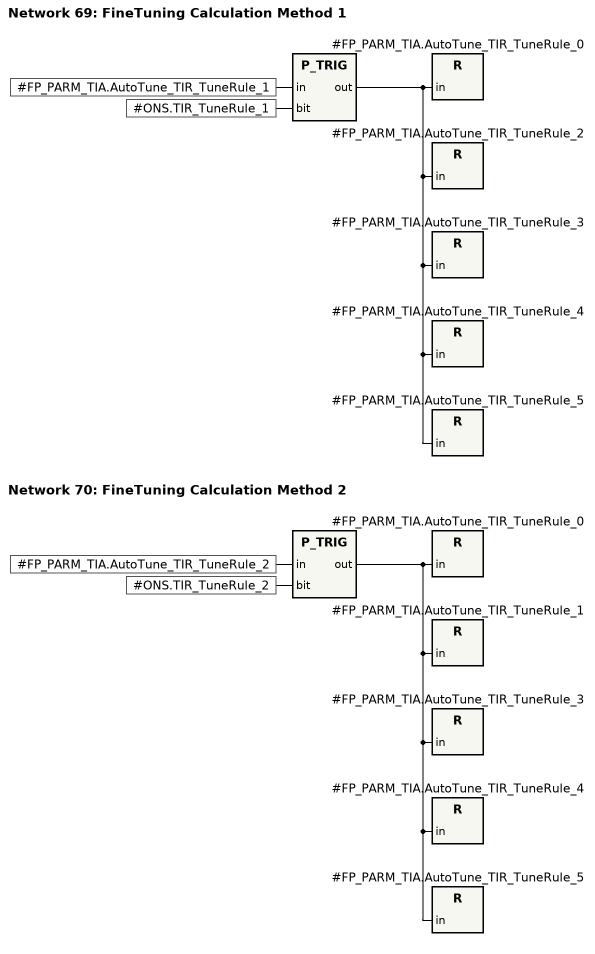
   #_w1 := #FP_PARM_TIA.AutoTune_TIR_TuneRule_1 AND NOT #ONS.TIR_TuneRule_1;   // rising edge
   #ONS.TIR_TuneRule_1 := #FP_PARM_TIA.AutoTune_TIR_TuneRule_1;
   IF #_w1 THEN
       #FP_PARM_TIA.AutoTune_TIR_TuneRule_0 := FALSE;
       #FP_PARM_TIA.AutoTune_TIR_TuneRule_2 := FALSE;
       #FP_PARM_TIA.AutoTune_TIR_TuneRule_3 := FALSE;
       #FP_PARM_TIA.AutoTune_TIR_TuneRule_4 := FALSE;
       #FP_PARM_TIA.AutoTune_TIR_TuneRule_5 := FALSE;
   END_IF;
END_REGION

REGION Network 70: FineTuning Calculation Method 2
   #_w1 := #FP_PARM_TIA.AutoTune_TIR_TuneRule_2 AND NOT #ONS.TIR_TuneRule_2;   // rising edge
   #ONS.TIR_TuneRule_2 := #FP_PARM_TIA.AutoTune_TIR_TuneRule_2;
   IF #_w1 THEN
       #FP_PARM_TIA.AutoTune_TIR_TuneRule_0 := FALSE;
       #FP_PARM_TIA.AutoTune_TIR_TuneRule_1 := FALSE;
       #FP_PARM_TIA.AutoTune_TIR_TuneRule_3 := FALSE;
       #FP_PARM_TIA.AutoTune_TIR_TuneRule_4 := FALSE;
       #FP_PARM_TIA.AutoTune_TIR_TuneRule_5 := FALSE;
   END_IF;
END_REGION

REGION Network 71: FineTuning Calculation Method 3
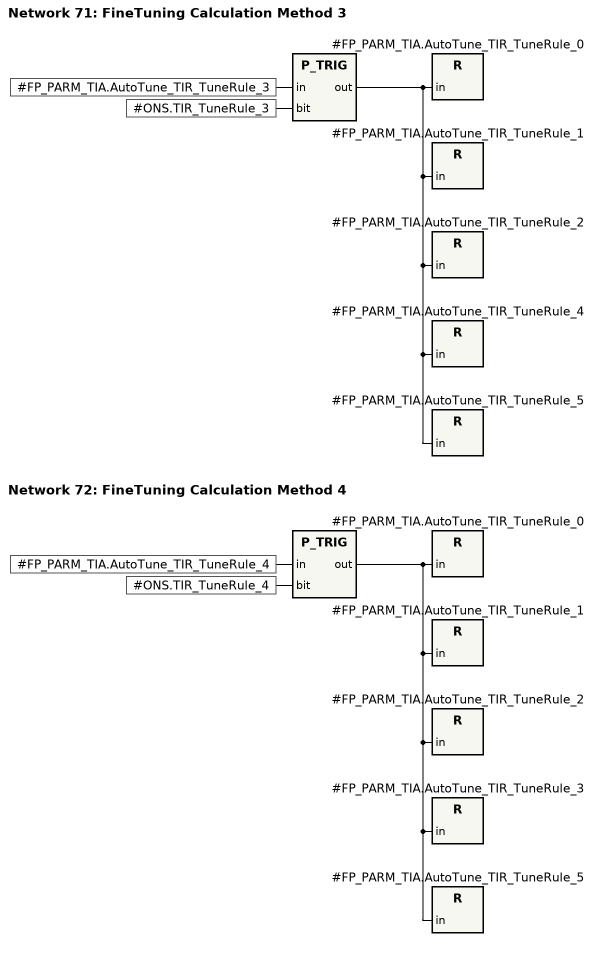
   #_w1 := #FP_PARM_TIA.AutoTune_TIR_TuneRule_3 AND NOT #ONS.TIR_TuneRule_3;   // rising edge
   #ONS.TIR_TuneRule_3 := #FP_PARM_TIA.AutoTune_TIR_TuneRule_3;
   IF #_w1 THEN
       #FP_PARM_TIA.AutoTune_TIR_TuneRule_0 := FALSE;
       #FP_PARM_TIA.AutoTune_TIR_TuneRule_1 := FALSE;
       #FP_PARM_TIA.AutoTune_TIR_TuneRule_2 := FALSE;
       #FP_PARM_TIA.AutoTune_TIR_TuneRule_4 := FALSE;
       #FP_PARM_TIA.AutoTune_TIR_TuneRule_5 := FALSE;
   END_IF;
END_REGION

REGION Network 72: FineTuning Calculation Method 4
   #_w1 := #FP_PARM_TIA.AutoTune_TIR_TuneRule_4 AND NOT #ONS.TIR_TuneRule_4;   // rising edge
   #ONS.TIR_TuneRule_4 := #FP_PARM_TIA.AutoTune_TIR_TuneRule_4;
   IF #_w1 THEN
       #FP_PARM_TIA.AutoTune_TIR_TuneRule_0 := FALSE;
       #FP_PARM_TIA.AutoTune_TIR_TuneRule_1 := FALSE;
       #FP_PARM_TIA.AutoTune_TIR_TuneRule_2 := FALSE;
       #FP_PARM_TIA.AutoTune_TIR_TuneRule_3 := FALSE;
       #FP_PARM_TIA.AutoTune_TIR_TuneRule_5 := FALSE;
   END_IF;
END_REGION

REGION Network 73: FineTuning Calculation Method 5
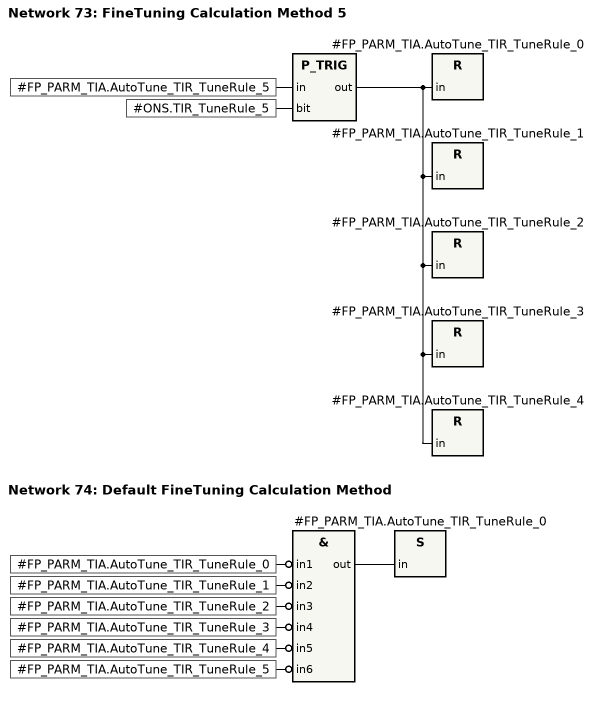
   #_w1 := #FP_PARM_TIA.AutoTune_TIR_TuneRule_5 AND NOT #ONS.TIR_TuneRule_5;   // rising edge
   #ONS.TIR_TuneRule_5 := #FP_PARM_TIA.AutoTune_TIR_TuneRule_5;
   IF #_w1 THEN
       #FP_PARM_TIA.AutoTune_TIR_TuneRule_0 := FALSE;
       #FP_PARM_TIA.AutoTune_TIR_TuneRule_1 := FALSE;
       #FP_PARM_TIA.AutoTune_TIR_TuneRule_2 := FALSE;
       #FP_PARM_TIA.AutoTune_TIR_TuneRule_3 := FALSE;
       #FP_PARM_TIA.AutoTune_TIR_TuneRule_4 := FALSE;
   END_IF;
END_REGION

REGION Network 74: Default FineTuning Calculation Method
   IF NOT #FP_PARM_TIA.AutoTune_TIR_TuneRule_0 AND NOT #FP_PARM_TIA.AutoTune_TIR_TuneRule_1 AND NOT #FP_PARM_TIA.AutoTune_TIR_TuneRule_2 AND NOT #FP_PARM_TIA.AutoTune_TIR_TuneRule_3 AND NOT #FP_PARM_TIA.AutoTune_TIR_TuneRule_4 AND NOT #FP_PARM_TIA.AutoTune_TIR_TuneRule_5 THEN
       #FP_PARM_TIA.AutoTune_TIR_TuneRule_0 := TRUE;
   END_IF;
END_REGION

REGION Network 75: AutoTune Parameterization
   // Build 002 - 04. Mar 2019 (RULA) : Typo in Auto tuning methods definition is corrected
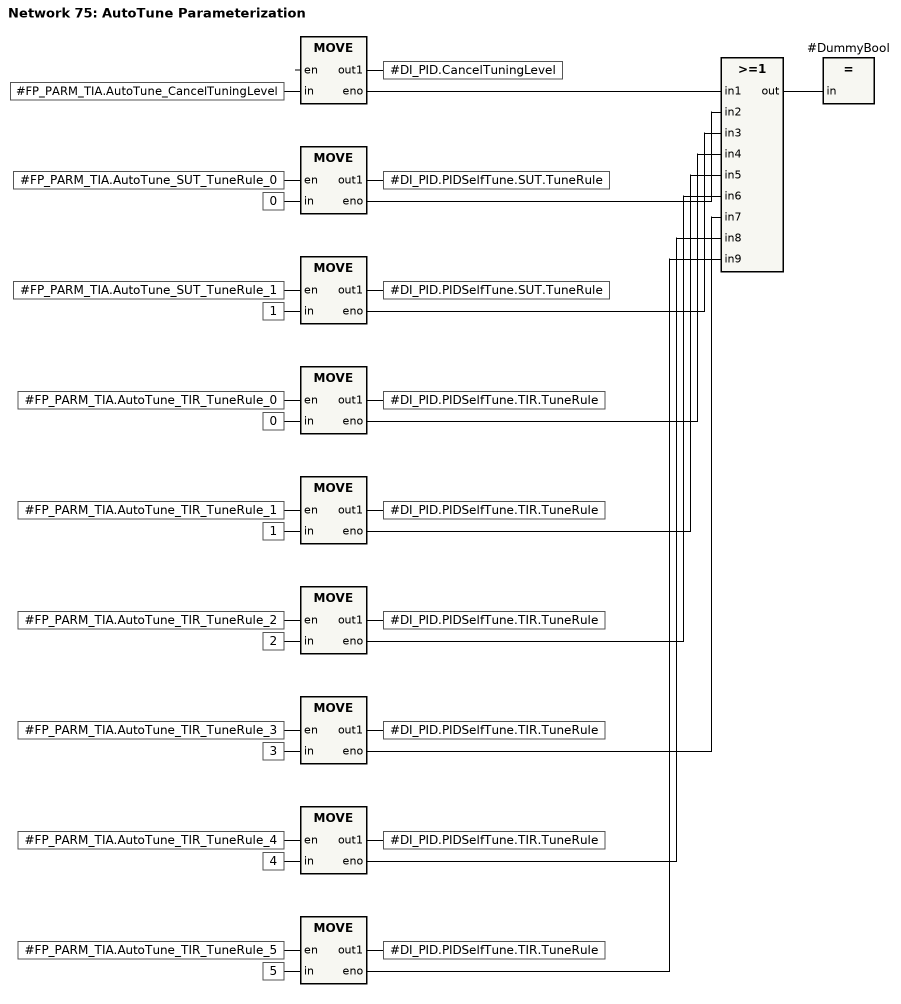
   #DI_PID.CancelTuningLevel := #FP_PARM_TIA.AutoTune_CancelTuningLevel;
   IF #FP_PARM_TIA.AutoTune_SUT_TuneRule_0 THEN #DI_PID.PIDSelfTune.SUT.TuneRule := 0; END_IF;
   IF #FP_PARM_TIA.AutoTune_SUT_TuneRule_1 THEN #DI_PID.PIDSelfTune.SUT.TuneRule := 1; END_IF;
   IF #FP_PARM_TIA.AutoTune_TIR_TuneRule_0 THEN #DI_PID.PIDSelfTune.TIR.TuneRule := 0; END_IF;
   IF #FP_PARM_TIA.AutoTune_TIR_TuneRule_1 THEN #DI_PID.PIDSelfTune.TIR.TuneRule := 1; END_IF;
   IF #FP_PARM_TIA.AutoTune_TIR_TuneRule_2 THEN #DI_PID.PIDSelfTune.TIR.TuneRule := 2; END_IF;
   IF #FP_PARM_TIA.AutoTune_TIR_TuneRule_3 THEN #DI_PID.PIDSelfTune.TIR.TuneRule := 3; END_IF;
   IF #FP_PARM_TIA.AutoTune_TIR_TuneRule_4 THEN #DI_PID.PIDSelfTune.TIR.TuneRule := 4; END_IF;
   IF #FP_PARM_TIA.AutoTune_TIR_TuneRule_5 THEN #DI_PID.PIDSelfTune.TIR.TuneRule := 5; END_IF;
   #DummyBool := TRUE OR #FP_PARM_TIA.AutoTune_SUT_TuneRule_0 OR #FP_PARM_TIA.AutoTune_SUT_TuneRule_1 OR #FP_PARM_TIA.AutoTune_TIR_TuneRule_0 OR #FP_PARM_TIA.AutoTune_TIR_TuneRule_1 OR #FP_PARM_TIA.AutoTune_TIR_TuneRule_2 OR #FP_PARM_TIA.AutoTune_TIR_TuneRule_3 OR #FP_PARM_TIA.AutoTune_TIR_TuneRule_4 OR #FP_PARM_TIA.AutoTune_TIR_TuneRule_5;
END_REGION

REGION Network 76: PreTuning Phase
   // 0: Initialize PreTuning
   // 100: Calculate Standard Deviation
   // 200: Find Point of Inflection
   // 9900: PreTuning Succesful
   // 1: PreTuning not Succesful
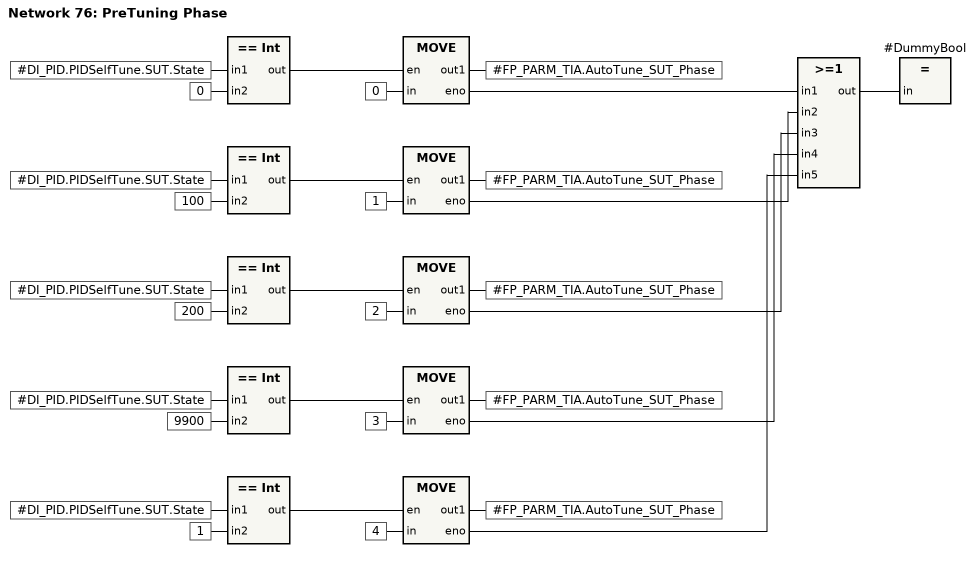
   #_w1 := #DI_PID.PIDSelfTune.SUT.State = 0;
   IF #_w1 THEN #FP_PARM_TIA.AutoTune_SUT_Phase := 0; END_IF;
   #_w2 := #DI_PID.PIDSelfTune.SUT.State = 100;
   IF #_w2 THEN #FP_PARM_TIA.AutoTune_SUT_Phase := 1; END_IF;
   #_w3 := #DI_PID.PIDSelfTune.SUT.State = 200;
   IF #_w3 THEN #FP_PARM_TIA.AutoTune_SUT_Phase := 2; END_IF;
   #_w4 := #DI_PID.PIDSelfTune.SUT.State = 9900;
   IF #_w4 THEN #FP_PARM_TIA.AutoTune_SUT_Phase := 3; END_IF;
   #_w5 := #DI_PID.PIDSelfTune.SUT.State = 1;
   IF #_w5 THEN #FP_PARM_TIA.AutoTune_SUT_Phase := 4; END_IF;
   #DummyBool := #_w1 OR #_w2 OR #_w3 OR #_w4 OR #_w5;
END_REGION

REGION Network 77: FineTuning Phase
   // -100: FineTuning not Possible.  PreTuning first
   // 0: Initialize FineTuning
   // 200:Calculate Standard Deviation
   // 300: Attempt to Reach Setpoint
   // 400: Attempt to Reach Sepoint with existing PID parameters
   // 500: Determine Oscillation and Calculate Parameters
   // 9900: FineTuning Success
   // 1: FineTuning not Succesful
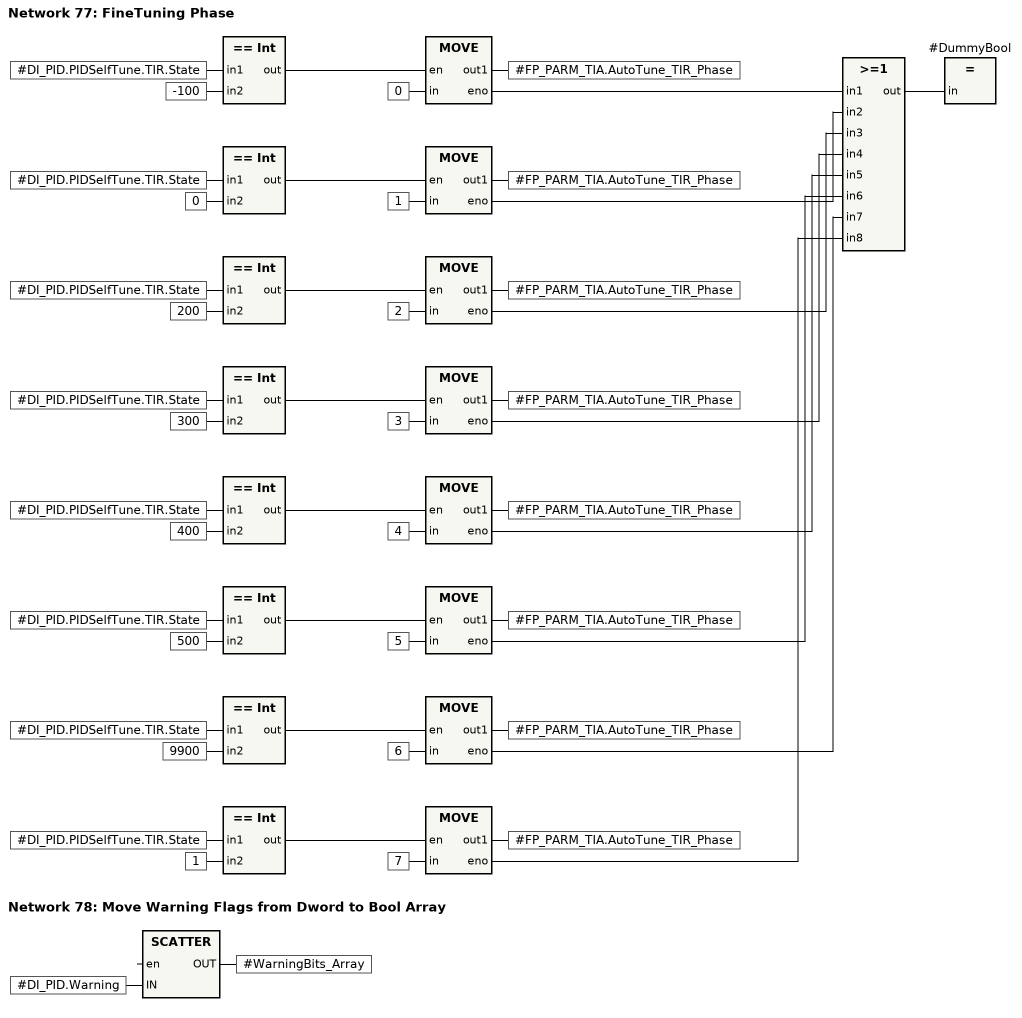
   #_w1 := #DI_PID.PIDSelfTune.TIR.State = (-100);
   IF #_w1 THEN #FP_PARM_TIA.AutoTune_TIR_Phase := 0; END_IF;
   #_w2 := #DI_PID.PIDSelfTune.TIR.State = 0;
   IF #_w2 THEN #FP_PARM_TIA.AutoTune_TIR_Phase := 1; END_IF;
   #_w3 := #DI_PID.PIDSelfTune.TIR.State = 200;
   IF #_w3 THEN #FP_PARM_TIA.AutoTune_TIR_Phase := 2; END_IF;
   #_w4 := #DI_PID.PIDSelfTune.TIR.State = 300;
   IF #_w4 THEN #FP_PARM_TIA.AutoTune_TIR_Phase := 3; END_IF;
   #_w5 := #DI_PID.PIDSelfTune.TIR.State = 400;
   IF #_w5 THEN #FP_PARM_TIA.AutoTune_TIR_Phase := 4; END_IF;
   #_w6 := #DI_PID.PIDSelfTune.TIR.State = 500;
   IF #_w6 THEN #FP_PARM_TIA.AutoTune_TIR_Phase := 5; END_IF;
   #_w7 := #DI_PID.PIDSelfTune.TIR.State = 9900;
   IF #_w7 THEN #FP_PARM_TIA.AutoTune_TIR_Phase := 6; END_IF;
   #_w8 := #DI_PID.PIDSelfTune.TIR.State = 1;
   IF #_w8 THEN #FP_PARM_TIA.AutoTune_TIR_Phase := 7; END_IF;
   #DummyBool := #_w1 OR #_w2 OR #_w3 OR #_w4 OR #_w5 OR #_w6 OR #_w7 OR #_w8;
END_REGION

REGION Network 78: Move Warning Flags from Dword to Bool Array
   SCATTER(IN := #DI_PID.Warning, OUT => #WarningBits_Array);
END_REGION

REGION Network 79: Warning Flags
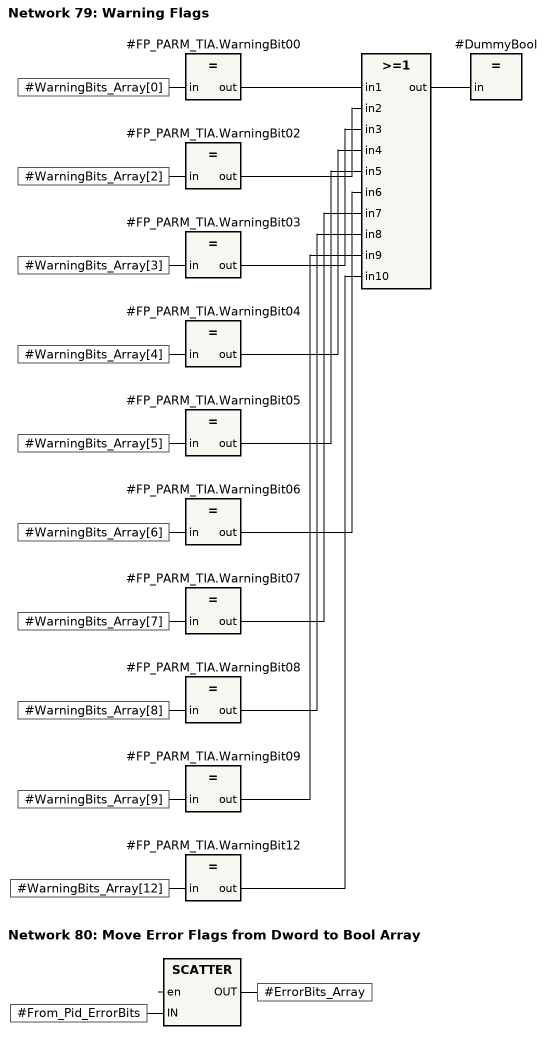
   #FP_PARM_TIA.WarningBit00 := #WarningBits_Array[0];
   #FP_PARM_TIA.WarningBit02 := #WarningBits_Array[2];
   #FP_PARM_TIA.WarningBit03 := #WarningBits_Array[3];
   #FP_PARM_TIA.WarningBit04 := #WarningBits_Array[4];
   #FP_PARM_TIA.WarningBit05 := #WarningBits_Array[5];
   #FP_PARM_TIA.WarningBit06 := #WarningBits_Array[6];
   #FP_PARM_TIA.WarningBit07 := #WarningBits_Array[7];
   #FP_PARM_TIA.WarningBit08 := #WarningBits_Array[8];
   #FP_PARM_TIA.WarningBit09 := #WarningBits_Array[9];
   #FP_PARM_TIA.WarningBit12 := #WarningBits_Array[12];
   #DummyBool := #WarningBits_Array[0] OR #WarningBits_Array[2] OR #WarningBits_Array[3] OR #WarningBits_Array[4] OR #WarningBits_Array[5] OR #WarningBits_Array[6] OR #WarningBits_Array[7] OR #WarningBits_Array[8] OR #WarningBits_Array[9] OR #WarningBits_Array[12];
END_REGION

REGION Network 80: Move Error Flags from Dword to Bool Array
   SCATTER(IN := #From_Pid_ErrorBits, OUT => #ErrorBits_Array);
END_REGION

REGION Network 81: Error Flags
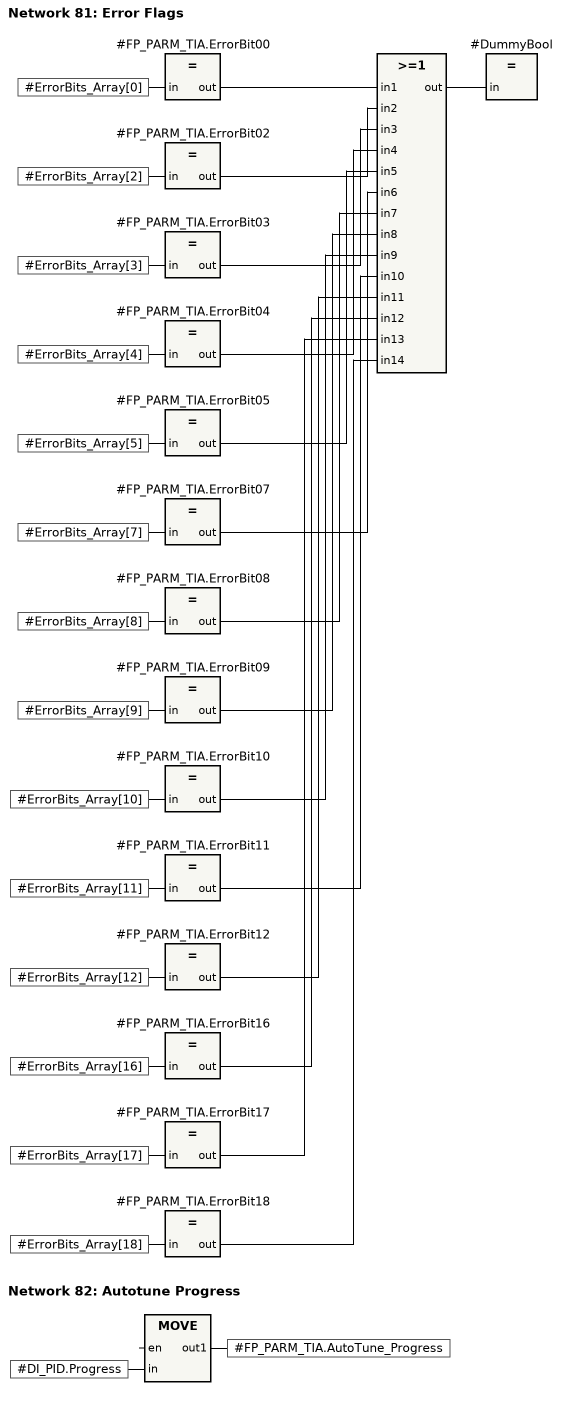
   #FP_PARM_TIA.ErrorBit00 := #ErrorBits_Array[0];
   #FP_PARM_TIA.ErrorBit02 := #ErrorBits_Array[2];
   #FP_PARM_TIA.ErrorBit03 := #ErrorBits_Array[3];
   #FP_PARM_TIA.ErrorBit04 := #ErrorBits_Array[4];
   #FP_PARM_TIA.ErrorBit05 := #ErrorBits_Array[5];
   #FP_PARM_TIA.ErrorBit07 := #ErrorBits_Array[7];
   #FP_PARM_TIA.ErrorBit08 := #ErrorBits_Array[8];
   #FP_PARM_TIA.ErrorBit09 := #ErrorBits_Array[9];
   #FP_PARM_TIA.ErrorBit10 := #ErrorBits_Array[10];
   #FP_PARM_TIA.ErrorBit11 := #ErrorBits_Array[11];
   #FP_PARM_TIA.ErrorBit12 := #ErrorBits_Array[12];
   #FP_PARM_TIA.ErrorBit16 := #ErrorBits_Array[16];
   #FP_PARM_TIA.ErrorBit17 := #ErrorBits_Array[17];
   #FP_PARM_TIA.ErrorBit18 := #ErrorBits_Array[18];
   #DummyBool := #ErrorBits_Array[0] OR #ErrorBits_Array[2] OR #ErrorBits_Array[3] OR #ErrorBits_Array[4] OR #ErrorBits_Array[5] OR #ErrorBits_Array[7] OR #ErrorBits_Array[8] OR #ErrorBits_Array[9] OR #ErrorBits_Array[10] OR #ErrorBits_Array[11] OR #ErrorBits_Array[12] OR #ErrorBits_Array[16] OR #ErrorBits_Array[17] OR #ErrorBits_Array[18];
END_REGION

REGION Network 82: Autotune Progress
   #FP_PARM_TIA.AutoTune_Progress := #DI_PID.Progress;
END_REGION

REGION Network 83: Update SPM Normalized
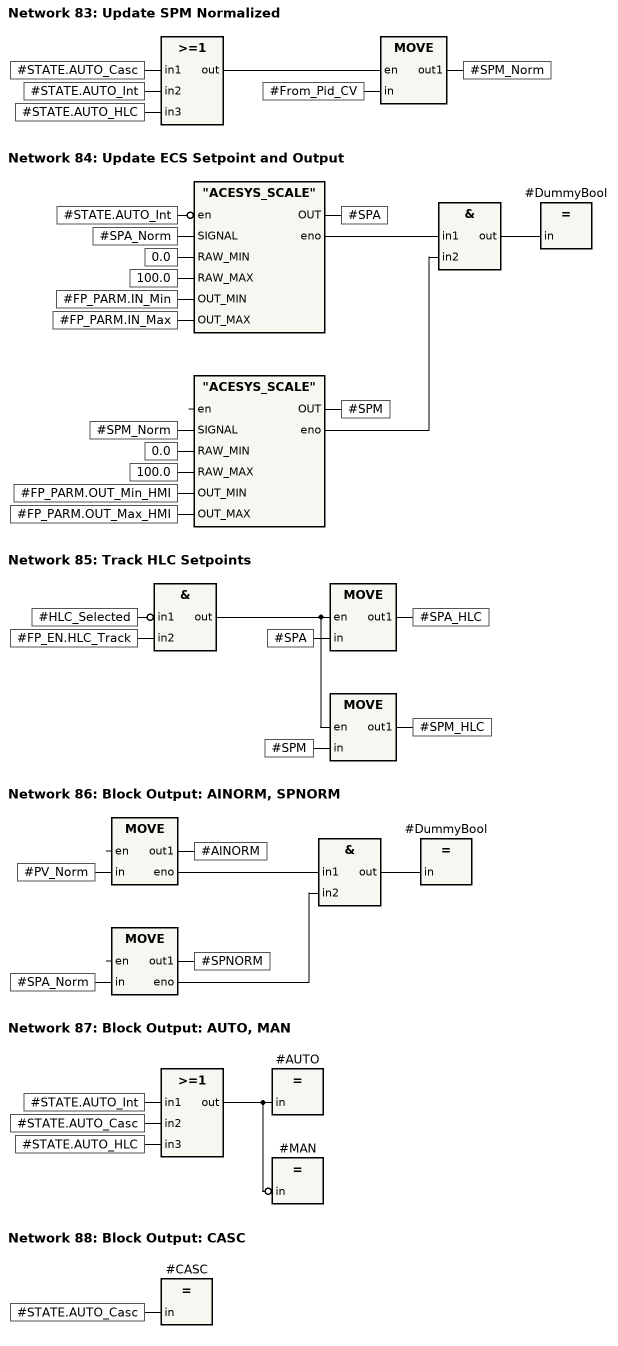
   IF #STATE.AUTO_Casc OR #STATE.AUTO_Int OR #STATE.AUTO_HLC THEN #SPM_Norm := #From_Pid_CV; END_IF;
END_REGION

REGION Network 84: Update ECS Setpoint and Output
   "ACESYS_SCALE"(EN := NOT #STATE.AUTO_Int,
                  SIGNAL := #SPA_Norm,
                  RAW_MIN := 0.0,
                  RAW_MAX := 100.0,
                  OUT_MIN := #FP_PARM.IN_Min,
                  OUT_MAX := #FP_PARM.IN_Max,
                  OUT => #SPA,
                  ENO => #_w1);
   "ACESYS_SCALE"(SIGNAL := #SPM_Norm,
                  RAW_MIN := 0.0,
                  RAW_MAX := 100.0,
                  OUT_MIN := #FP_PARM.OUT_Min_HMI,
                  OUT_MAX := #FP_PARM.OUT_Max_HMI,
                  OUT => #SPM,
                  ENO => #_w2);
   #DummyBool := #_w1 AND #_w2;
END_REGION

REGION Network 85: Track HLC Setpoints
   IF NOT #HLC_Selected AND #FP_EN.HLC_Track THEN
       #SPA_HLC := #SPA;
       #SPM_HLC := #SPM;
   END_IF;
END_REGION

REGION Network 86: Block Output: AINORM, SPNORM
   // >>>>> BLOCK OUTPUT <<<<<
   // ENO of a box is taken as its EN; it also drops when the box reports an error
   #AINORM := #PV_Norm;
   #SPNORM := #SPA_Norm;
   #DummyBool := TRUE;
END_REGION

REGION Network 87: Block Output: AUTO, MAN
   #AUTO := #STATE.AUTO_Int OR #STATE.AUTO_Casc OR #STATE.AUTO_HLC;
   #MAN := NOT #AUTO;
END_REGION

REGION Network 88: Block Output: CASC
   #CASC := #STATE.AUTO_Casc;
END_REGION

REGION Network 89: Normalized Error
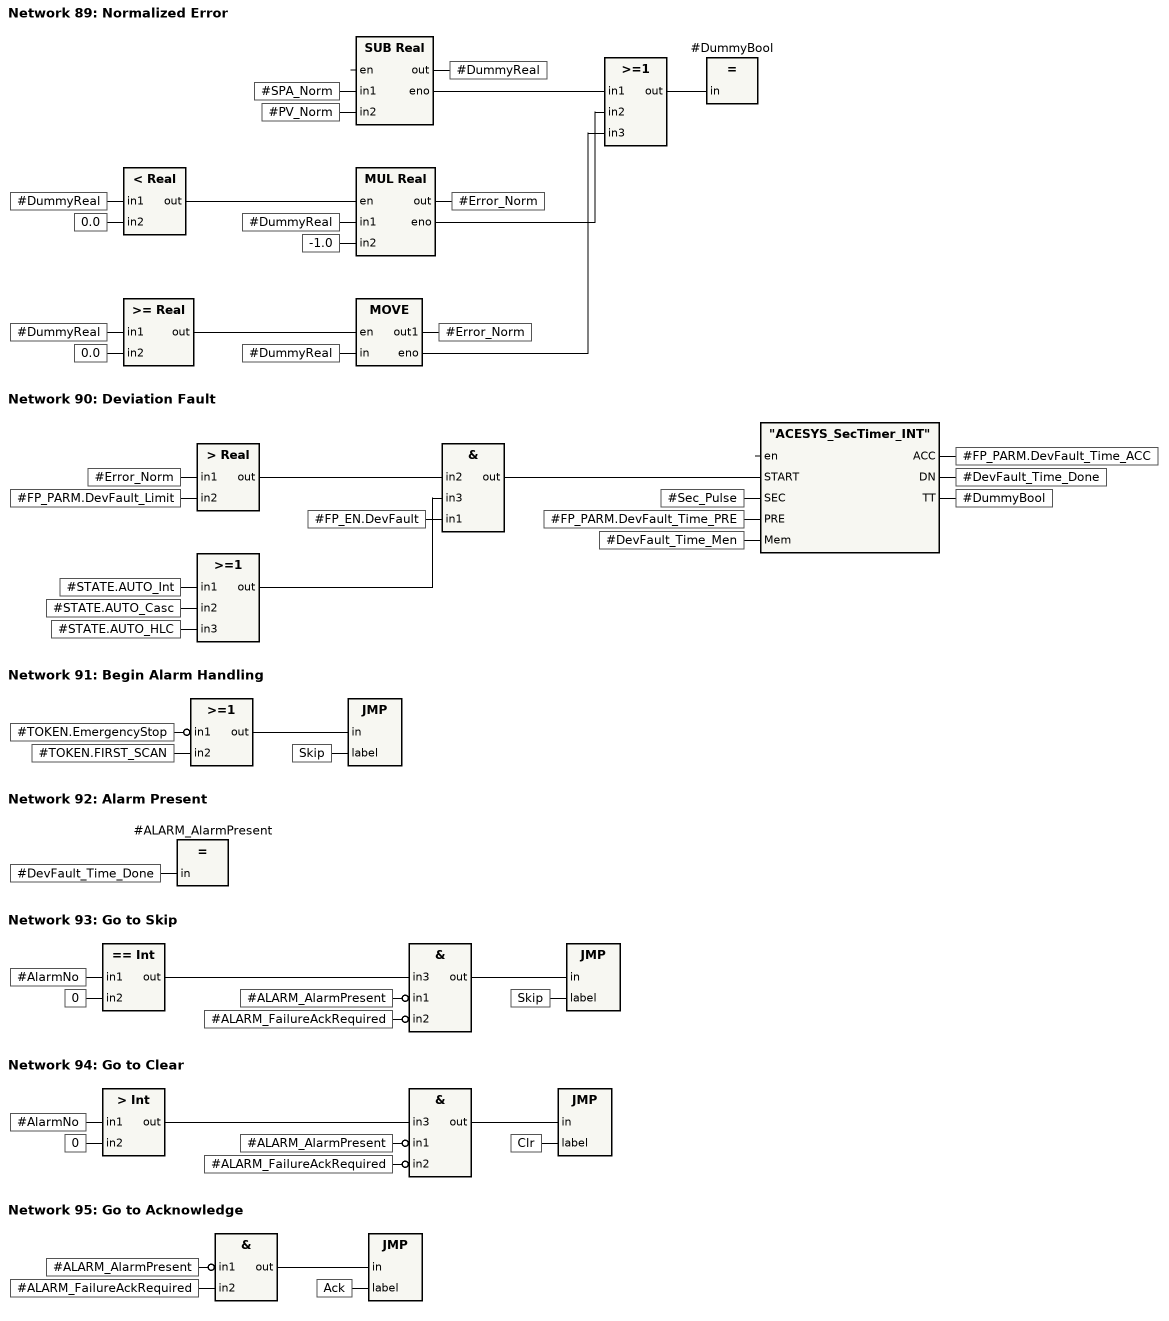
   #DummyReal := #SPA_Norm - #PV_Norm;
   #_w1 := #DummyReal < 0.0;
   IF #_w1 THEN #Error_Norm := #DummyReal * (-1.0); END_IF;
   #_w2 := #DummyReal >= 0.0;
   IF #_w2 THEN #Error_Norm := #DummyReal; END_IF;
   #DummyBool := TRUE OR #_w1 OR #_w2;
END_REGION

REGION Network 90: Deviation Fault
   // >>>>> DEVIATION FAULT <<<<<
   "ACESYS_SecTimer_INT"(START := (#Error_Norm > #FP_PARM.DevFault_Limit) AND (#STATE.AUTO_Int OR #STATE.AUTO_Casc OR #STATE.AUTO_HLC) AND #FP_EN.DevFault,
                         SEC := #Sec_Pulse,
                         PRE := #FP_PARM.DevFault_Time_PRE,
                         Mem := #DevFault_Time_Men,
                         ACC => #FP_PARM.DevFault_Time_ACC,
                         DN => #DevFault_Time_Done,
                         TT => #DummyBool);
END_REGION

REGION Network 91: Begin Alarm Handling
   // >>>>> ALARM HANDLING <<<<<
   IF NOT #TOKEN.EmergencyStop OR #TOKEN.FIRST_SCAN THEN GOTO Skip; END_IF;
END_REGION

REGION Network 92: Alarm Present
   #ALARM_AlarmPresent := #DevFault_Time_Done;
END_REGION

REGION Network 93: Go to Skip
   IF (#AlarmNo = 0) AND NOT #ALARM_AlarmPresent AND NOT #ALARM_FailureAckRequired THEN GOTO Skip; END_IF;
END_REGION

REGION Network 94: Go to Clear
   IF (#AlarmNo > 0) AND NOT #ALARM_AlarmPresent AND NOT #ALARM_FailureAckRequired THEN GOTO Clr; END_IF;
END_REGION

REGION Network 95: Go to Acknowledge
   IF NOT #ALARM_AlarmPresent AND #ALARM_FailureAckRequired THEN GOTO Ack; END_IF;
END_REGION

REGION Network 96: Alarm: Deviation Failure
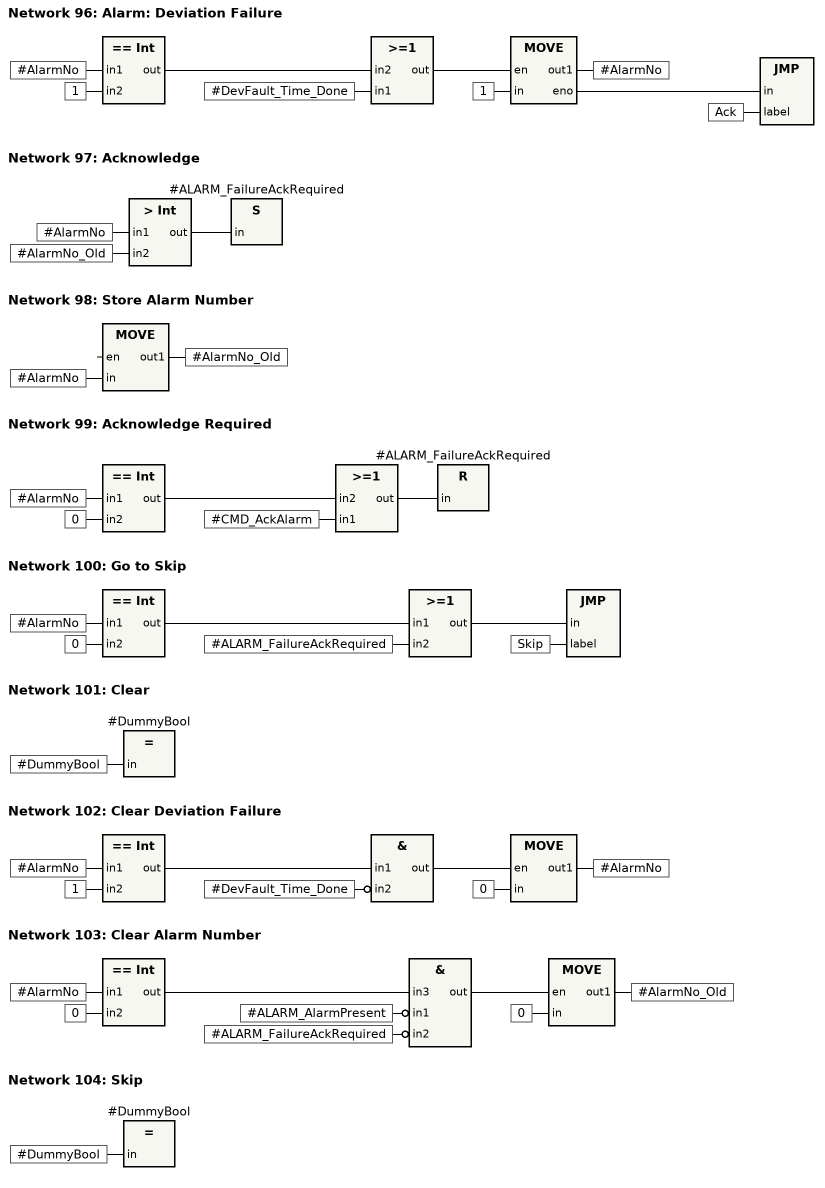
   // ENO of a box is taken as its EN; it also drops when the box reports an error
   #_w1 := (#AlarmNo = 1) OR #DevFault_Time_Done;
   IF #_w1 THEN
       #AlarmNo := 1;
       GOTO Ack;
   END_IF;
END_REGION

REGION Network 97: Acknowledge
   // ***Alarm Acknowledge***
   Ack:
   IF #AlarmNo > #AlarmNo_Old THEN #ALARM_FailureAckRequired := TRUE; END_IF;
END_REGION

REGION Network 98: Store Alarm Number
   #AlarmNo_Old := #AlarmNo;
END_REGION

REGION Network 99: Acknowledge Required
   IF (#AlarmNo = 0) OR #CMD_AckAlarm THEN #ALARM_FailureAckRequired := FALSE; END_IF;
END_REGION

REGION Network 100: Go to Skip
   IF (#AlarmNo = 0) OR #ALARM_FailureAckRequired THEN GOTO Skip; END_IF;
END_REGION

REGION Network 101: Clear
   Clr:
   #DummyBool := #DummyBool;
END_REGION

REGION Network 102: Clear Deviation Failure
   IF (#AlarmNo = 1) AND NOT #DevFault_Time_Done THEN #AlarmNo := 0; END_IF;
END_REGION

REGION Network 103: Clear Alarm Number
   IF (#AlarmNo = 0) AND NOT #ALARM_AlarmPresent AND NOT #ALARM_FailureAckRequired THEN
       #AlarmNo_Old := 0;
   END_IF;
END_REGION

REGION Network 104: Skip
   Skip:
   #DummyBool := #DummyBool;
END_REGION

REGION Network 105: Extended MSW
   // >>>> EXTENDED MSW to HMI <<<<<
   // 
   // Build 003 : 27. Jan. 2016 (FKP) : Network for #MSW.EXT.Operation changed from 
   //                                   AND- to OR-gate
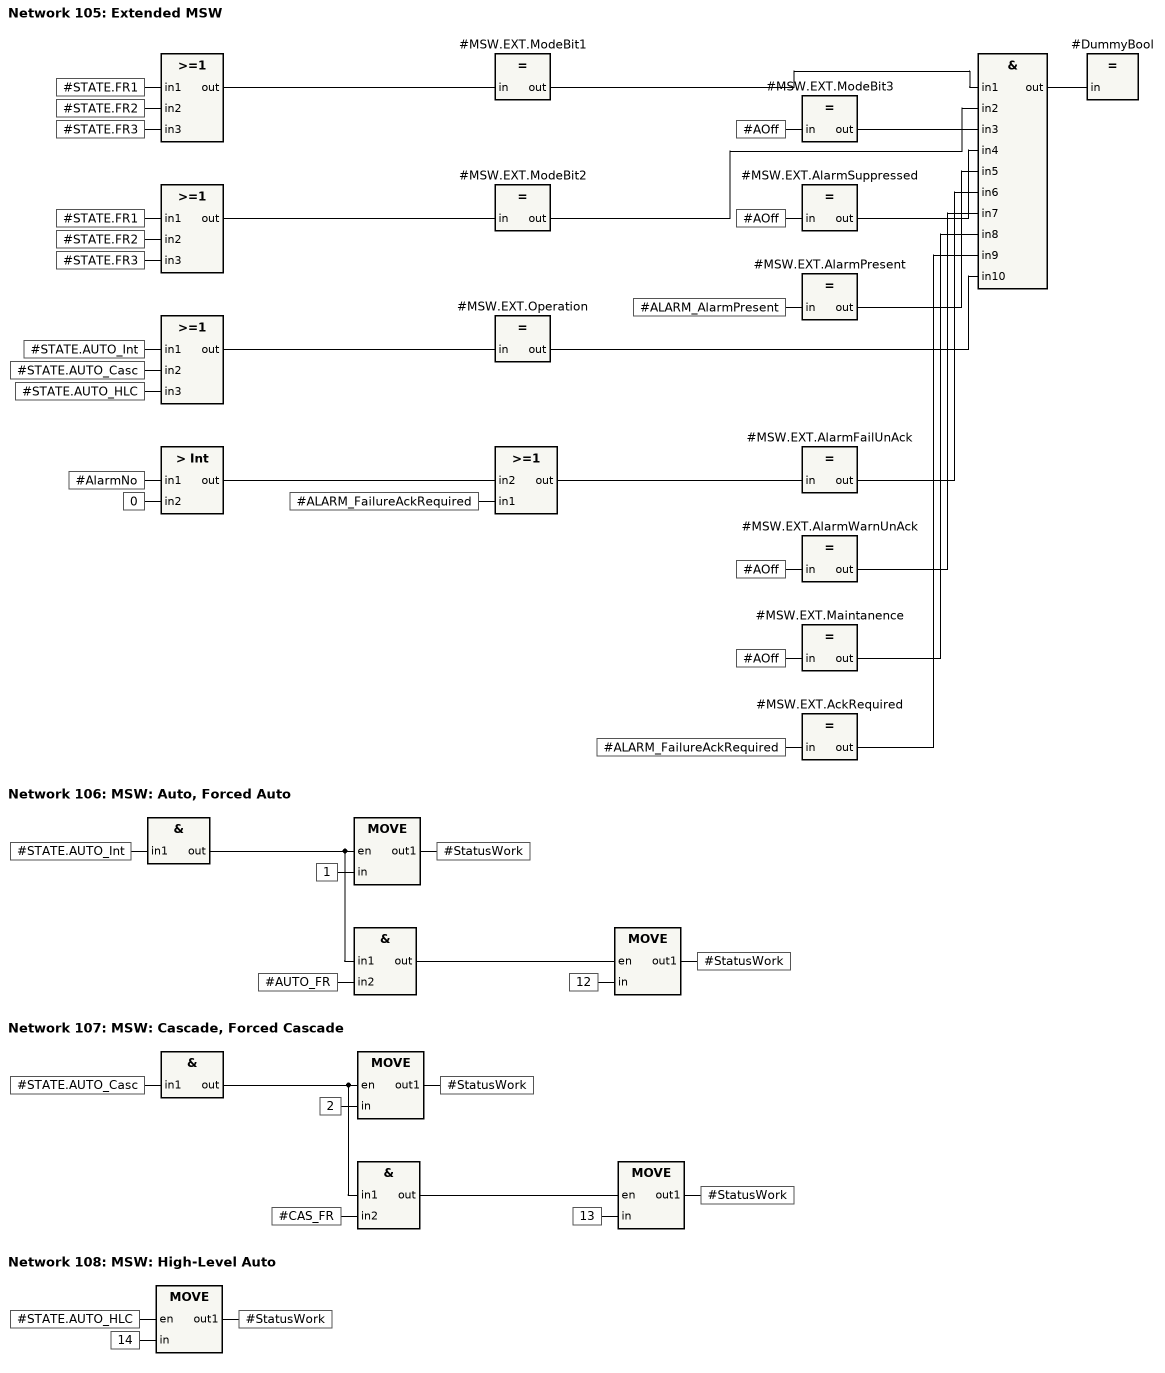
   #MSW.EXT.ModeBit1 := #STATE.FR1 OR #STATE.FR2 OR #STATE.FR3;
   #MSW.EXT.ModeBit2 := #STATE.FR1 OR #STATE.FR2 OR #STATE.FR3;
   #MSW.EXT.ModeBit3 := #AOff;
   #MSW.EXT.AlarmSuppressed := #AOff;
   #MSW.EXT.AlarmPresent := #ALARM_AlarmPresent;
   #MSW.EXT.AlarmFailUnAck := (#AlarmNo > 0) OR #ALARM_FailureAckRequired;
   #MSW.EXT.AlarmWarnUnAck := #AOff;
   #MSW.EXT.Maintanence := #AOff;
   #MSW.EXT.AckRequired := #ALARM_FailureAckRequired;
   #MSW.EXT.Operation := #STATE.AUTO_Int OR #STATE.AUTO_Casc OR #STATE.AUTO_HLC;
   #DummyBool := #MSW.EXT.ModeBit1 AND #MSW.EXT.ModeBit2 AND #AOff AND #AOff AND #ALARM_AlarmPresent AND #MSW.EXT.AlarmFailUnAck AND #AOff AND #AOff AND #ALARM_FailureAckRequired AND #MSW.EXT.Operation;
END_REGION

REGION Network 106: MSW: Auto, Forced Auto
   IF #STATE.AUTO_Int THEN #StatusWork := 1; END_IF;
   IF #STATE.AUTO_Int AND #AUTO_FR THEN #StatusWork := 12; END_IF;
END_REGION

REGION Network 107: MSW: Cascade, Forced Cascade
   IF #STATE.AUTO_Casc THEN #StatusWork := 2; END_IF;
   IF #STATE.AUTO_Casc AND #CAS_FR THEN #StatusWork := 13; END_IF;
END_REGION

REGION Network 108: MSW: High-Level Auto
   IF #STATE.AUTO_HLC THEN #StatusWork := 14; END_IF;
END_REGION

REGION Network 109: MSW: Manual, Forced Manual
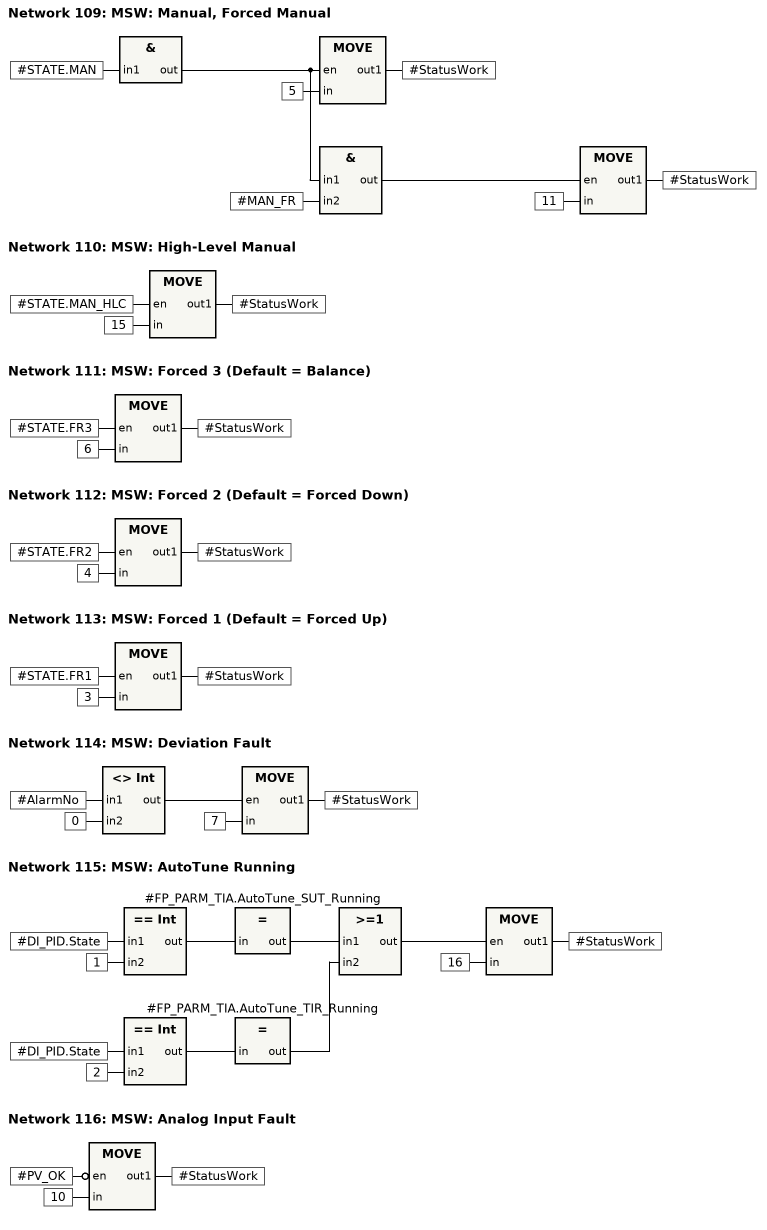
   IF #STATE.MAN THEN #StatusWork := 5; END_IF;
   IF #STATE.MAN AND #MAN_FR THEN #StatusWork := 11; END_IF;
END_REGION

REGION Network 110: MSW: High-Level Manual
   IF #STATE.MAN_HLC THEN #StatusWork := 15; END_IF;
END_REGION

REGION Network 111: MSW: Forced 3 (Default = Balance)
   IF #STATE.FR3 THEN #StatusWork := 6; END_IF;
END_REGION

REGION Network 112: MSW: Forced 2 (Default = Forced Down)
   IF #STATE.FR2 THEN #StatusWork := 4; END_IF;
END_REGION

REGION Network 113: MSW: Forced 1 (Default = Forced Up)
   IF #STATE.FR1 THEN #StatusWork := 3; END_IF;
END_REGION

REGION Network 114: MSW: Deviation Fault
   IF #AlarmNo <> 0 THEN #StatusWork := 7; END_IF;
END_REGION

REGION Network 115: MSW: AutoTune Running
   #FP_PARM_TIA.AutoTune_SUT_Running := #DI_PID.State = 1;
   #FP_PARM_TIA.AutoTune_TIR_Running := #DI_PID.State = 2;
   IF #FP_PARM_TIA.AutoTune_SUT_Running OR #FP_PARM_TIA.AutoTune_TIR_Running THEN #StatusWork := 16; END_IF;
END_REGION

REGION Network 116: MSW: Analog Input Fault
   IF NOT #PV_OK THEN #StatusWork := 10; END_IF;
END_REGION

REGION Network 117: Update Internal MSW and Timestamp
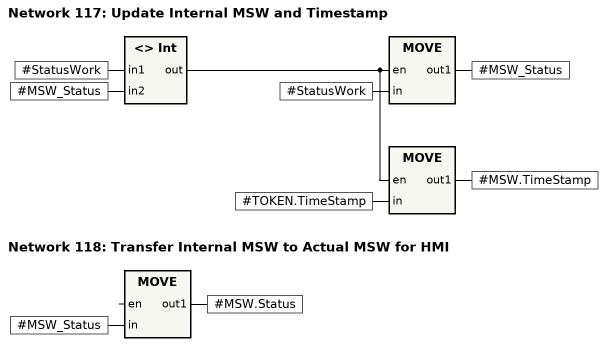
   #_w1 := #StatusWork <> #MSW_Status;
   IF #_w1 THEN
       #MSW_Status := #StatusWork;
       #MSW.TimeStamp := #TOKEN.TimeStamp;
   END_IF;
END_REGION

REGION Network 118: Transfer Internal MSW to Actual MSW for HMI
   #MSW.Status := #MSW_Status;
END_REGION
END_FUNCTION_BLOCK

FUNCTION_BLOCK "ACESYS_HLC"   // FB221, FBD
TITLE = ACESYS V8.0 - Build 001 - HIGH LEVEL CONTROL
{ S7_Optimized_Access := 'FALSE' }
AUTHOR : FLSmidth
FAMILY : ACESYS
NAME : HLC
VERSION : 8.0
   VAR_INPUT
      DEPT_LINK : "ACESYS_DEPT_LINK";   // Unit Number
      CCA1 : Bool := TRUE;   // Computer Control Accept Group 01-05
      CCA2 : Bool := TRUE;   // Computer Control Accept Group 06-10
      GRP_01_RDY : Bool := TRUE;   // Group 01 Ready
      GRP_02_RDY : Bool := TRUE;   // Group 02 Ready
      GRP_03_RDY : Bool := TRUE;   // Group 03 Ready
      GRP_04_RDY : Bool := TRUE;   // Group 04 Ready
      GRP_05_RDY : Bool := TRUE;   // Group 05 Ready
      GRP_06_RDY : Bool := TRUE;   // Group 06 Ready
      GRP_07_RDY : Bool := TRUE;   // Group 07 Ready
      GRP_08_RDY : Bool := TRUE;   // Group 08 Ready
      GRP_09_RDY : Bool := TRUE;   // Group 09 Ready
      GRP_10_RDY : Bool := TRUE;   // Group 10 Ready
   END_VAR
   VAR_OUTPUT
      HLC_LINK : "ACESYS_HLC_LINK";
      MSW : "ACESYS_HMI_STAT_32T";
   END_VAR
   VAR_IN_OUT
      KA : Bool;   // Keep Alive - Watchdog supervision
      GRP_01_EN : Bool;   // Enable Group 01
      GRP_02_EN : Bool;   // Enable Group 02
      GRP_03_EN : Bool;   // Enable Group 03
      GRP_04_EN : Bool;   // Enable Group 04
      GRP_05_EN : Bool;   // Enable Group 05
      GRP_06_EN : Bool;   // Enable Group 06
      GRP_07_EN : Bool;   // Enable Group 07
      GRP_08_EN : Bool;   // Enable Group 08
      GRP_09_EN : Bool;   // Enable Group 09
      GRP_10_EN : Bool;   // Enable Group 10
   END_VAR
   VAR
      BlockInfo : Struct
         Ace_Version : Int;   // Acesys Block Version Number
         Ace_BuildNo : Int;   // Acesys Block Build Number
         DB_Number : Int;   // Block Instance DB Number
      END_STRUCT;
      FP_CMD : Struct   // Faceplate Commands
         Spare_08 : Bool;
         Spare_09 : Bool;
         Spare_10 : Bool;
         Spare_11 : Bool;
         Spare_12 : Bool;
         Spare_13 : Bool;
         Spare_14 : Bool;
         AckAlarm : Bool;   // Alarm Acknowledge
         Spare_00 : Bool;
         Spare_01 : Bool;
         Spare_02 : Bool;
         Spare_03 : Bool;
         Spare_04 : Bool;
         Spare_05 : Bool;
         Spare_06 : Bool;
         Spare_07 : Bool;
      END_STRUCT;
      FP_SEL : Struct
         GRP_01 : Bool;
         GRP_02 : Bool;
         GRP_03 : Bool;
         GRP_04 : Bool;
         GRP_05 : Bool;
         GRP_06 : Bool;
         GRP_07 : Bool;
         GRP_08 : Bool;
         GRP_09 : Bool;
         GRP_10 : Bool;
         KA_Alarm : Bool;   // Select KA Supervision
         CCA1_Alarm : Bool;   // Select CCA Supervision HLC Group 01-05
         CCA2_Alarm : Bool;   // Select CCA Supervision HLC Group 06-10
         Spare3 : Bool;
         Spare2 : Bool;
         Spare1 : Bool;
      END_STRUCT;
      FP_EN : Struct
         Clear_Sel_CCA : Bool;   // Clear Selections when CCA Faults
         Clear_Sel_KA : Bool;   // Clear Selections when KA Fault
         Spare14 : Bool;
         Spare13 : Bool;
         Spare12 : Bool;
         Spare11 : Bool;
         Spare10 : Bool;
         Spare09 : Bool;
         Spare08 : Bool;
         Spare07 : Bool;
         Spare06 : Bool;
         Spare05 : Bool;
         Spare04 : Bool;
         Spare03 : Bool;
         Spare02 : Bool;
         Spare01 : Bool;
      END_STRUCT;
      FP_PARM : Struct
         KA_Time_Actual : Int;   // Keep Alive remaining time
         KA_Time_Setp : Int := 60;   // Keep Alive Setpoint
      END_STRUCT;
      ONS : Struct
         ONS_Off : Array[1..16] of Bool;
         ONS_On : Array[1..16] of Bool;
         OFF_01 : Bool;
         OFF_02 : Bool;
         OFF_03 : Bool;
         OFF_04 : Bool;
         OFF_05 : Bool;
         OFF_06 : Bool;
         OFF_07 : Bool;
         OFF_08 : Bool;
         OFF_09 : Bool;
         OFF_10 : Bool;
         ON_01 : Bool;
         ON_02 : Bool;
         ON_03 : Bool;
         ON_04 : Bool;
         ON_05 : Bool;
         ON_06 : Bool;
         ON_07 : Bool;
         ON_08 : Bool;
         ON_09 : Bool;
         ON_10 : Bool;
      END_STRUCT;
      KA_Time_Memory : Int;   // Keep Alive memory
      StatusToEcs : Int;
      ALARM_AlarmPresent : Bool;
      ALARM_FailureAckRequired : Bool;
      CMD_AckAlarm : Bool;
      StatusWork : Int;   // Internal Status Word
      AlarmNo : Int;
      AlarmNo_Old : Int;
      MSW_Status_Trans : Int;
   END_VAR
   VAR_TEMP
      Aon : Bool;
      Aoff : Bool;
      DummyBool : Bool;
      Acknowledge : Bool;   // Alarm Acknowledge
      KeepAliveTimeDone : Bool;
      TrigAlarm_KA : Bool;
      TrigAlarm_CCA1 : Bool;
      TrigAlarm_CCA2 : Bool;
   END_VAR
   VAR_TEMP   // added for the SCL form of the ladder/FBD networks
      _w1 : Bool;
   END_VAR
BEGIN

REGION Network 1: Always On
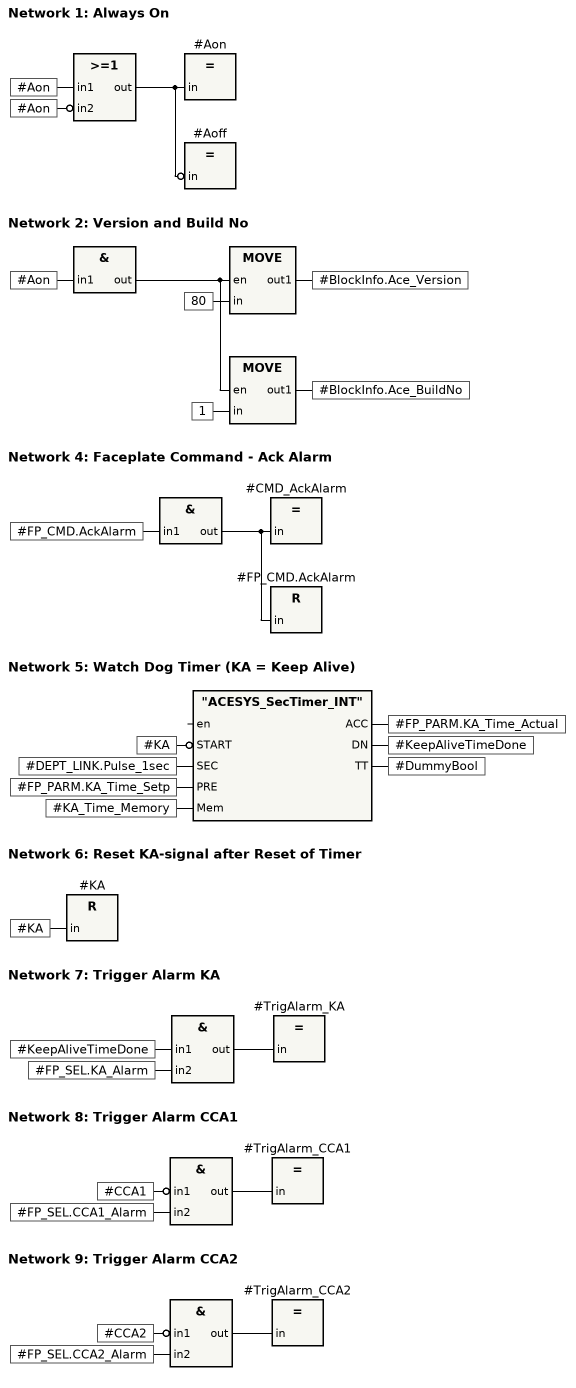
   #Aon := #Aon OR NOT #Aon;
   #Aoff := NOT #Aon;
END_REGION

REGION Network 2: Version and Build No
   IF #Aon THEN
       #BlockInfo.Ace_Version := 80;
       #BlockInfo.Ace_BuildNo := 1;
   END_IF;
END_REGION

REGION Network 3 (STL): Instance DB Number to Faceplate
         L     DINO;
         T     #BlockInfo.DB_Number;
END_REGION

REGION Network 4: Faceplate Command - Ack Alarm
   #CMD_AckAlarm := #FP_CMD.AckAlarm;
   IF #FP_CMD.AckAlarm THEN #FP_CMD.AckAlarm := FALSE; END_IF;
END_REGION

REGION Network 5: Watch Dog Timer (KA = Keep Alive)
   "ACESYS_SecTimer_INT"(START := NOT #KA,
                         SEC := #DEPT_LINK.Pulse_1sec,
                         PRE := #FP_PARM.KA_Time_Setp,
                         Mem := #KA_Time_Memory,
                         ACC => #FP_PARM.KA_Time_Actual,
                         DN => #KeepAliveTimeDone,
                         TT => #DummyBool);
END_REGION

REGION Network 6: Reset KA-signal after Reset of Timer
   IF #KA THEN #KA := FALSE; END_IF;
END_REGION

REGION Network 7: Trigger Alarm KA
   #TrigAlarm_KA := #KeepAliveTimeDone AND #FP_SEL.KA_Alarm;
END_REGION

REGION Network 8: Trigger Alarm CCA1
   #TrigAlarm_CCA1 := NOT #CCA1 AND #FP_SEL.CCA1_Alarm;
END_REGION

REGION Network 9: Trigger Alarm CCA2
   #TrigAlarm_CCA2 := NOT #CCA2 AND #FP_SEL.CCA2_Alarm;
END_REGION

REGION Network 10: If Intput is changed, Update Faceplate Parameters - Sel GRP01
   // >>>>> SELECT <<<<<
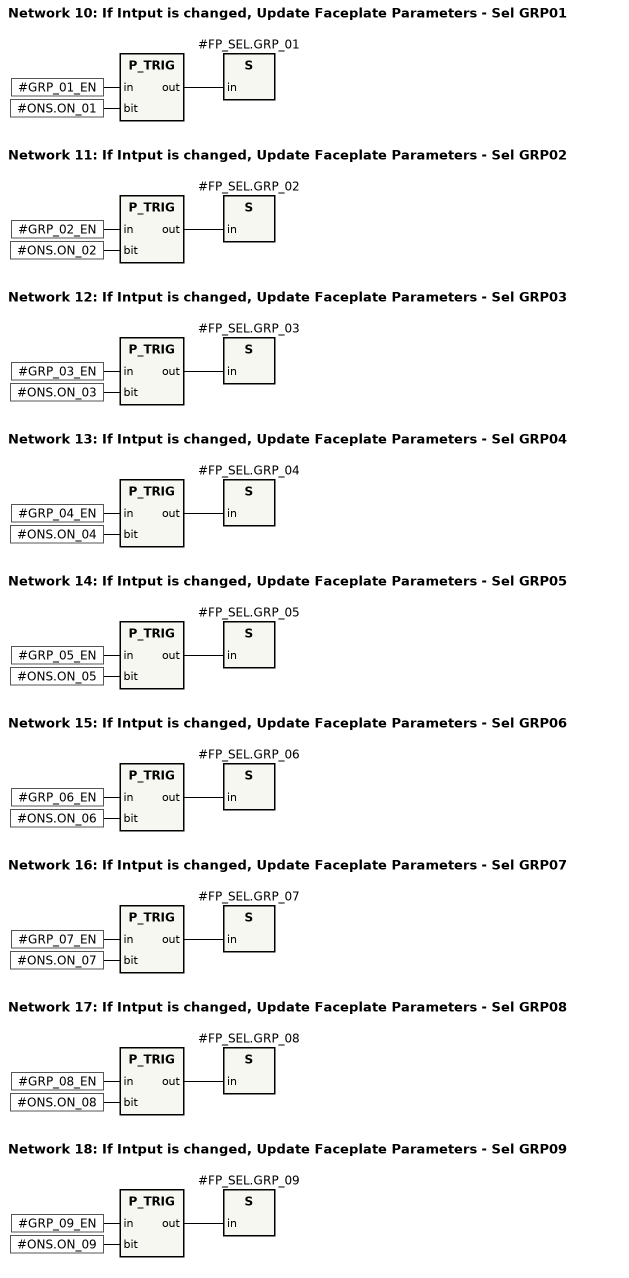
   #_w1 := #GRP_01_EN AND NOT #ONS.ON_01;   // rising edge
   #ONS.ON_01 := #GRP_01_EN;
   IF #_w1 THEN #FP_SEL.GRP_01 := TRUE; END_IF;
END_REGION

REGION Network 11: If Intput is changed, Update Faceplate Parameters - Sel GRP02
   #_w1 := #GRP_02_EN AND NOT #ONS.ON_02;   // rising edge
   #ONS.ON_02 := #GRP_02_EN;
   IF #_w1 THEN #FP_SEL.GRP_02 := TRUE; END_IF;
END_REGION

REGION Network 12: If Intput is changed, Update Faceplate Parameters - Sel GRP03
   #_w1 := #GRP_03_EN AND NOT #ONS.ON_03;   // rising edge
   #ONS.ON_03 := #GRP_03_EN;
   IF #_w1 THEN #FP_SEL.GRP_03 := TRUE; END_IF;
END_REGION

REGION Network 13: If Intput is changed, Update Faceplate Parameters - Sel GRP04
   #_w1 := #GRP_04_EN AND NOT #ONS.ON_04;   // rising edge
   #ONS.ON_04 := #GRP_04_EN;
   IF #_w1 THEN #FP_SEL.GRP_04 := TRUE; END_IF;
END_REGION

REGION Network 14: If Intput is changed, Update Faceplate Parameters - Sel GRP05
   #_w1 := #GRP_05_EN AND NOT #ONS.ON_05;   // rising edge
   #ONS.ON_05 := #GRP_05_EN;
   IF #_w1 THEN #FP_SEL.GRP_05 := TRUE; END_IF;
END_REGION

REGION Network 15: If Intput is changed, Update Faceplate Parameters - Sel GRP06
   #_w1 := #GRP_06_EN AND NOT #ONS.ON_06;   // rising edge
   #ONS.ON_06 := #GRP_06_EN;
   IF #_w1 THEN #FP_SEL.GRP_06 := TRUE; END_IF;
END_REGION

REGION Network 16: If Intput is changed, Update Faceplate Parameters - Sel GRP07
   #_w1 := #GRP_07_EN AND NOT #ONS.ON_07;   // rising edge
   #ONS.ON_07 := #GRP_07_EN;
   IF #_w1 THEN #FP_SEL.GRP_07 := TRUE; END_IF;
END_REGION

REGION Network 17: If Intput is changed, Update Faceplate Parameters - Sel GRP08
   #_w1 := #GRP_08_EN AND NOT #ONS.ON_08;   // rising edge
   #ONS.ON_08 := #GRP_08_EN;
   IF #_w1 THEN #FP_SEL.GRP_08 := TRUE; END_IF;
END_REGION

REGION Network 18: If Intput is changed, Update Faceplate Parameters - Sel GRP09
   #_w1 := #GRP_09_EN AND NOT #ONS.ON_09;   // rising edge
   #ONS.ON_09 := #GRP_09_EN;
   IF #_w1 THEN #FP_SEL.GRP_09 := TRUE; END_IF;
END_REGION

REGION Network 19: If Intput is changed, Update Faceplate Parameters - Sel GRP10
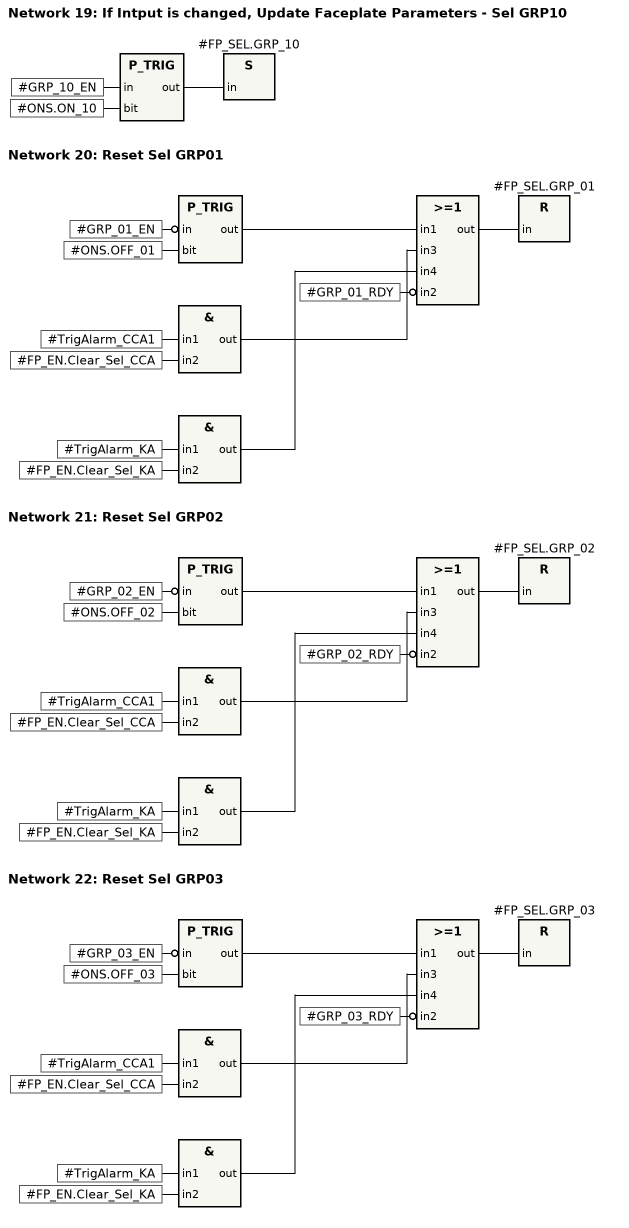
   #_w1 := #GRP_10_EN AND NOT #ONS.ON_10;   // rising edge
   #ONS.ON_10 := #GRP_10_EN;
   IF #_w1 THEN #FP_SEL.GRP_10 := TRUE; END_IF;
END_REGION

REGION Network 20: Reset Sel GRP01
   #_w1 := NOT #GRP_01_EN AND NOT #ONS.OFF_01;   // rising edge
   #ONS.OFF_01 := NOT #GRP_01_EN;
   IF #_w1 OR (#TrigAlarm_CCA1 AND #FP_EN.Clear_Sel_CCA) OR (#TrigAlarm_KA AND #FP_EN.Clear_Sel_KA) OR NOT #GRP_01_RDY THEN
       #FP_SEL.GRP_01 := FALSE;
   END_IF;
END_REGION

REGION Network 21: Reset Sel GRP02
   #_w1 := NOT #GRP_02_EN AND NOT #ONS.OFF_02;   // rising edge
   #ONS.OFF_02 := NOT #GRP_02_EN;
   IF #_w1 OR (#TrigAlarm_CCA1 AND #FP_EN.Clear_Sel_CCA) OR (#TrigAlarm_KA AND #FP_EN.Clear_Sel_KA) OR NOT #GRP_02_RDY THEN
       #FP_SEL.GRP_02 := FALSE;
   END_IF;
END_REGION

REGION Network 22: Reset Sel GRP03
   #_w1 := NOT #GRP_03_EN AND NOT #ONS.OFF_03;   // rising edge
   #ONS.OFF_03 := NOT #GRP_03_EN;
   IF #_w1 OR (#TrigAlarm_CCA1 AND #FP_EN.Clear_Sel_CCA) OR (#TrigAlarm_KA AND #FP_EN.Clear_Sel_KA) OR NOT #GRP_03_RDY THEN
       #FP_SEL.GRP_03 := FALSE;
   END_IF;
END_REGION

REGION Network 23: Reset Sel GRP04
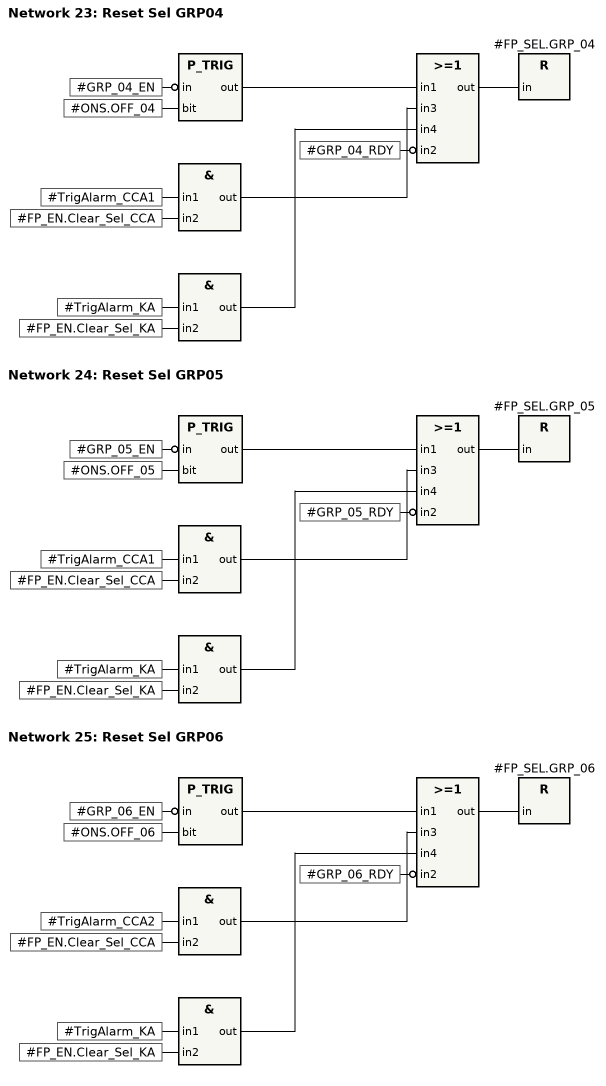
   #_w1 := NOT #GRP_04_EN AND NOT #ONS.OFF_04;   // rising edge
   #ONS.OFF_04 := NOT #GRP_04_EN;
   IF #_w1 OR (#TrigAlarm_CCA1 AND #FP_EN.Clear_Sel_CCA) OR (#TrigAlarm_KA AND #FP_EN.Clear_Sel_KA) OR NOT #GRP_04_RDY THEN
       #FP_SEL.GRP_04 := FALSE;
   END_IF;
END_REGION

REGION Network 24: Reset Sel GRP05
   #_w1 := NOT #GRP_05_EN AND NOT #ONS.OFF_05;   // rising edge
   #ONS.OFF_05 := NOT #GRP_05_EN;
   IF #_w1 OR (#TrigAlarm_CCA1 AND #FP_EN.Clear_Sel_CCA) OR (#TrigAlarm_KA AND #FP_EN.Clear_Sel_KA) OR NOT #GRP_05_RDY THEN
       #FP_SEL.GRP_05 := FALSE;
   END_IF;
END_REGION

REGION Network 25: Reset Sel GRP06
   #_w1 := NOT #GRP_06_EN AND NOT #ONS.OFF_06;   // rising edge
   #ONS.OFF_06 := NOT #GRP_06_EN;
   IF #_w1 OR (#TrigAlarm_CCA2 AND #FP_EN.Clear_Sel_CCA) OR (#TrigAlarm_KA AND #FP_EN.Clear_Sel_KA) OR NOT #GRP_06_RDY THEN
       #FP_SEL.GRP_06 := FALSE;
   END_IF;
END_REGION

REGION Network 26: Reset Sel GRP07
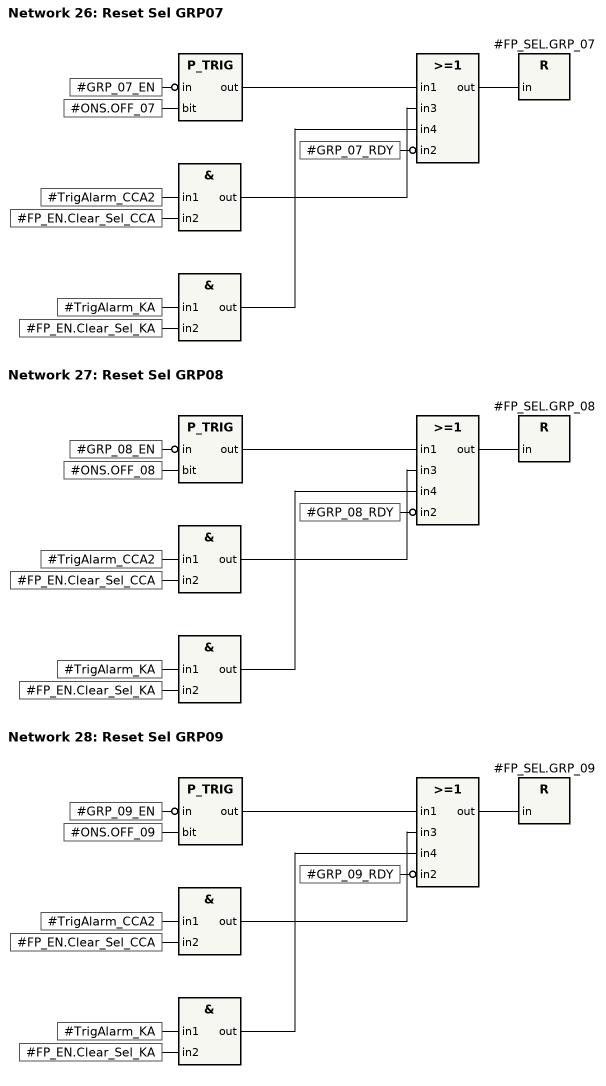
   #_w1 := NOT #GRP_07_EN AND NOT #ONS.OFF_07;   // rising edge
   #ONS.OFF_07 := NOT #GRP_07_EN;
   IF #_w1 OR (#TrigAlarm_CCA2 AND #FP_EN.Clear_Sel_CCA) OR (#TrigAlarm_KA AND #FP_EN.Clear_Sel_KA) OR NOT #GRP_07_RDY THEN
       #FP_SEL.GRP_07 := FALSE;
   END_IF;
END_REGION

REGION Network 27: Reset Sel GRP08
   #_w1 := NOT #GRP_08_EN AND NOT #ONS.OFF_08;   // rising edge
   #ONS.OFF_08 := NOT #GRP_08_EN;
   IF #_w1 OR (#TrigAlarm_CCA2 AND #FP_EN.Clear_Sel_CCA) OR (#TrigAlarm_KA AND #FP_EN.Clear_Sel_KA) OR NOT #GRP_08_RDY THEN
       #FP_SEL.GRP_08 := FALSE;
   END_IF;
END_REGION

REGION Network 28: Reset Sel GRP09
   #_w1 := NOT #GRP_09_EN AND NOT #ONS.OFF_09;   // rising edge
   #ONS.OFF_09 := NOT #GRP_09_EN;
   IF #_w1 OR (#TrigAlarm_CCA2 AND #FP_EN.Clear_Sel_CCA) OR (#TrigAlarm_KA AND #FP_EN.Clear_Sel_KA) OR NOT #GRP_09_RDY THEN
       #FP_SEL.GRP_09 := FALSE;
   END_IF;
END_REGION

REGION Network 29: Reset Sel GRP10
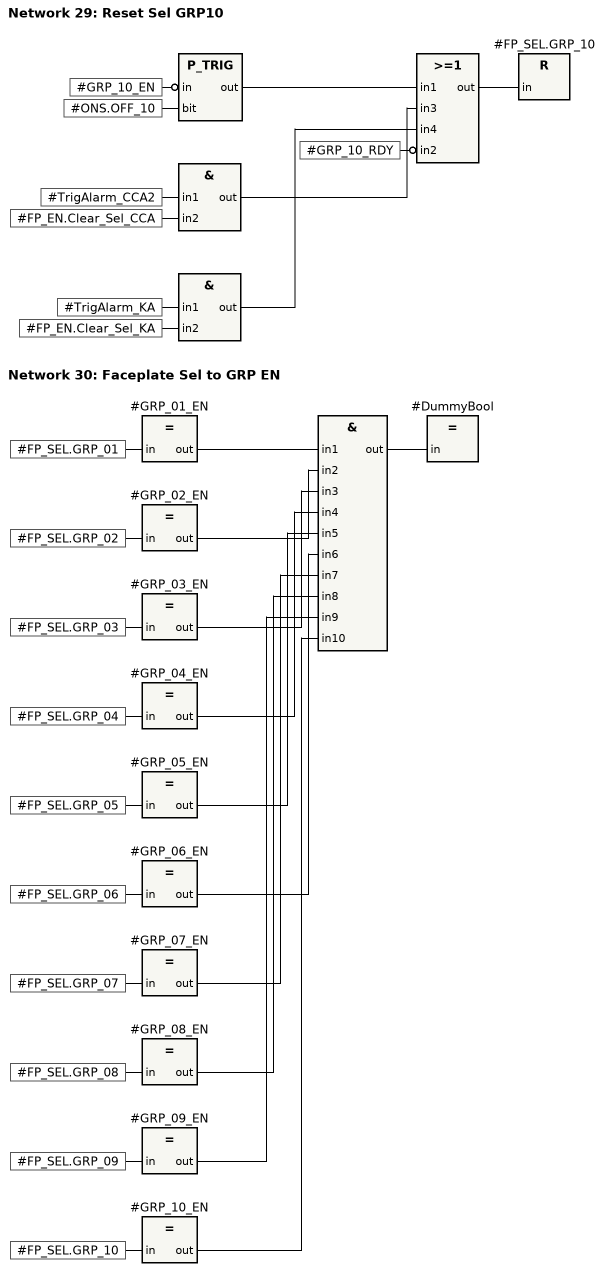
   #_w1 := NOT #GRP_10_EN AND NOT #ONS.OFF_10;   // rising edge
   #ONS.OFF_10 := NOT #GRP_10_EN;
   IF #_w1 OR (#TrigAlarm_CCA2 AND #FP_EN.Clear_Sel_CCA) OR (#TrigAlarm_KA AND #FP_EN.Clear_Sel_KA) OR NOT #GRP_10_RDY THEN
       #FP_SEL.GRP_10 := FALSE;
   END_IF;
END_REGION

REGION Network 30: Faceplate Sel to GRP EN
   #GRP_01_EN := #FP_SEL.GRP_01;
   #GRP_02_EN := #FP_SEL.GRP_02;
   #GRP_03_EN := #FP_SEL.GRP_03;
   #GRP_04_EN := #FP_SEL.GRP_04;
   #GRP_05_EN := #FP_SEL.GRP_05;
   #GRP_06_EN := #FP_SEL.GRP_06;
   #GRP_07_EN := #FP_SEL.GRP_07;
   #GRP_08_EN := #FP_SEL.GRP_08;
   #GRP_09_EN := #FP_SEL.GRP_09;
   #GRP_10_EN := #FP_SEL.GRP_10;
   #DummyBool := #FP_SEL.GRP_01 AND #FP_SEL.GRP_02 AND #FP_SEL.GRP_03 AND #FP_SEL.GRP_04 AND #FP_SEL.GRP_05 AND #FP_SEL.GRP_06 AND #FP_SEL.GRP_07 AND #FP_SEL.GRP_08 AND #FP_SEL.GRP_09 AND #FP_SEL.GRP_10;
END_REGION

REGION Network 31: Output to Group 01-05
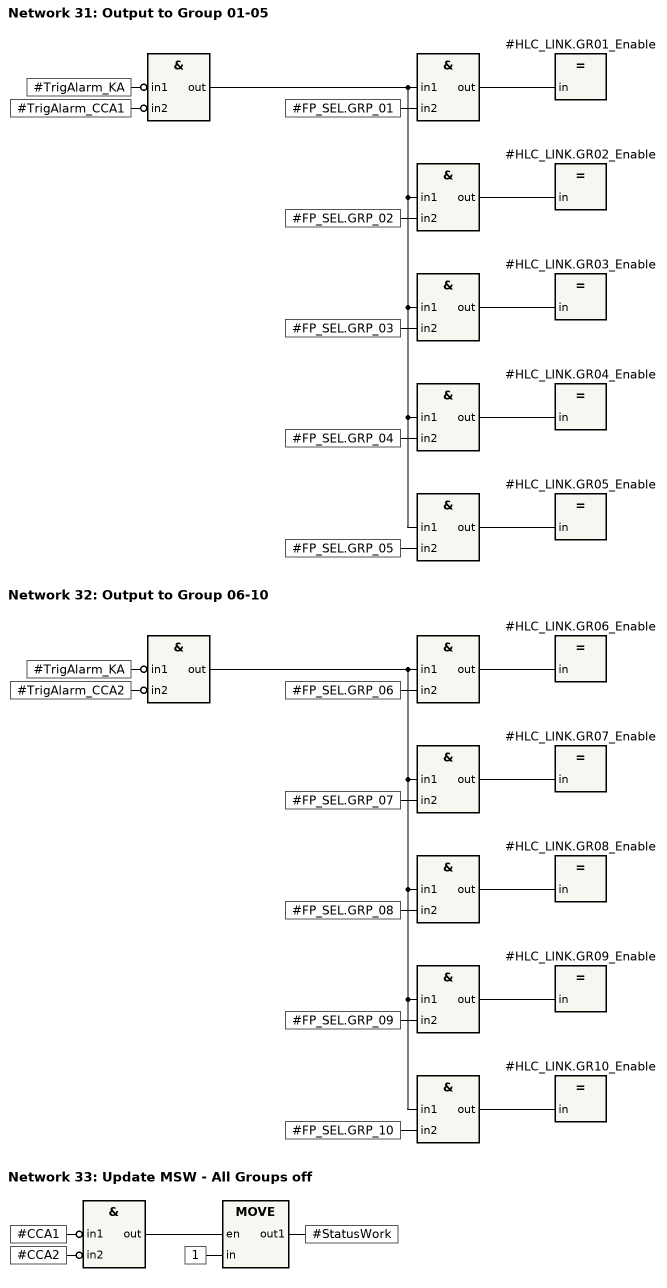
   #_w1 := NOT #TrigAlarm_KA AND NOT #TrigAlarm_CCA1;
   #HLC_LINK.GR01_Enable := #_w1 AND #FP_SEL.GRP_01;
   #HLC_LINK.GR02_Enable := #_w1 AND #FP_SEL.GRP_02;
   #HLC_LINK.GR03_Enable := #_w1 AND #FP_SEL.GRP_03;
   #HLC_LINK.GR04_Enable := #_w1 AND #FP_SEL.GRP_04;
   #HLC_LINK.GR05_Enable := #_w1 AND #FP_SEL.GRP_05;
END_REGION

REGION Network 32: Output to Group 06-10
   #_w1 := NOT #TrigAlarm_KA AND NOT #TrigAlarm_CCA2;
   #HLC_LINK.GR06_Enable := #_w1 AND #FP_SEL.GRP_06;
   #HLC_LINK.GR07_Enable := #_w1 AND #FP_SEL.GRP_07;
   #HLC_LINK.GR08_Enable := #_w1 AND #FP_SEL.GRP_08;
   #HLC_LINK.GR09_Enable := #_w1 AND #FP_SEL.GRP_09;
   #HLC_LINK.GR10_Enable := #_w1 AND #FP_SEL.GRP_10;
END_REGION

REGION Network 33: Update MSW - All Groups off
   IF NOT #CCA1 AND NOT #CCA2 THEN #StatusWork := 1; END_IF;
END_REGION

REGION Network 34: Update MSW - Group 01-05 On
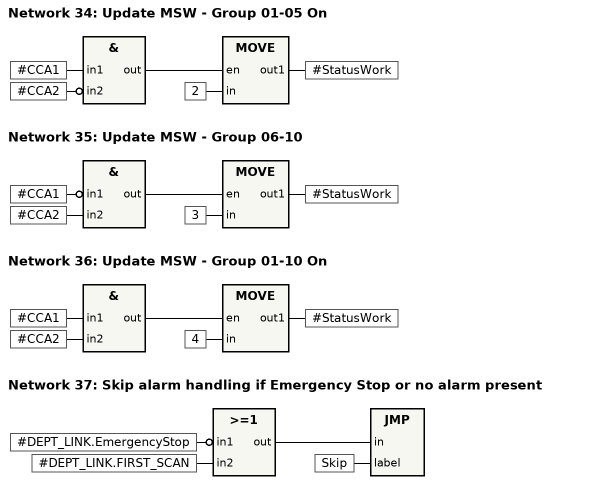
   IF #CCA1 AND NOT #CCA2 THEN #StatusWork := 2; END_IF;
END_REGION

REGION Network 35: Update MSW - Group 06-10
   IF NOT #CCA1 AND #CCA2 THEN #StatusWork := 3; END_IF;
END_REGION

REGION Network 36: Update MSW - Group 01-10 On
   IF #CCA1 AND #CCA2 THEN #StatusWork := 4; END_IF;
END_REGION

REGION Network 37: Skip alarm handling if Emergency Stop or no alarm present
   // Skip = Skip Alarm
   IF NOT #DEPT_LINK.EmergencyStop OR #DEPT_LINK.FIRST_SCAN THEN GOTO Skip; END_IF;
END_REGION

REGION Network 38: Alarm Present
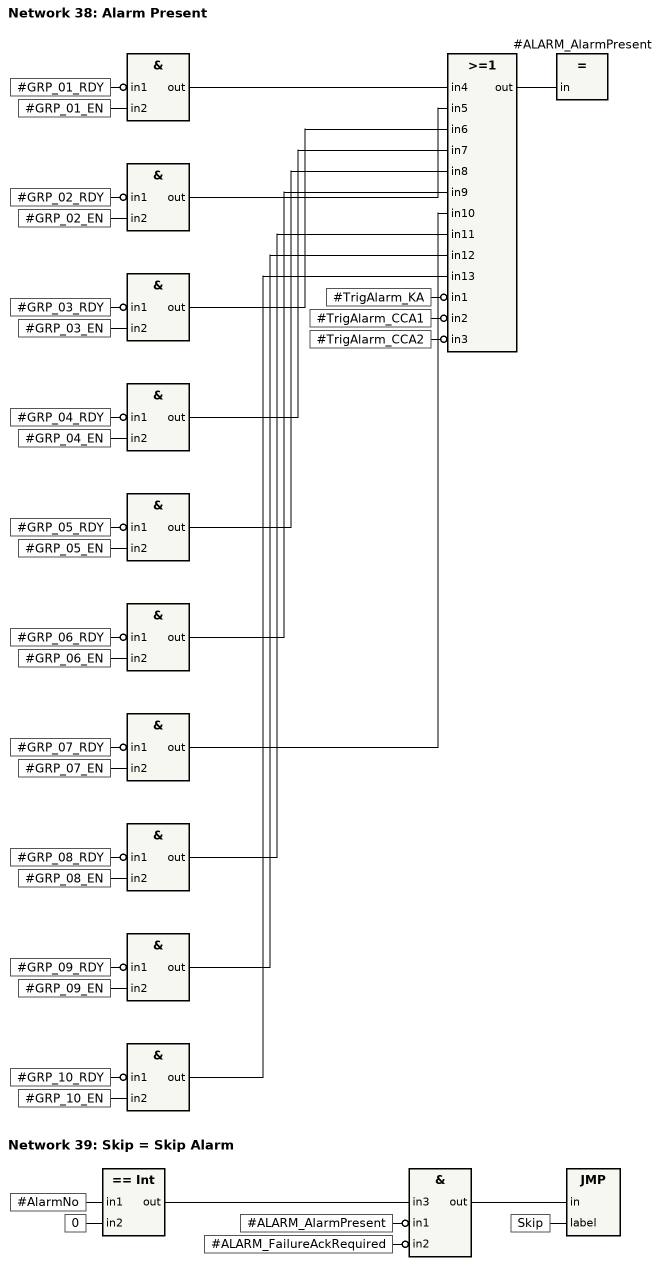
   #ALARM_AlarmPresent := (NOT #GRP_01_RDY AND #GRP_01_EN) OR (NOT #GRP_02_RDY AND #GRP_02_EN) OR (NOT #GRP_03_RDY AND #GRP_03_EN) OR (NOT #GRP_04_RDY AND #GRP_04_EN) OR (NOT #GRP_05_RDY AND #GRP_05_EN) OR (NOT #GRP_06_RDY AND #GRP_06_EN) OR (NOT #GRP_07_RDY AND #GRP_07_EN) OR (NOT #GRP_08_RDY AND #GRP_08_EN) OR (NOT #GRP_09_RDY AND #GRP_09_EN) OR (NOT #GRP_10_RDY AND #GRP_10_EN) OR NOT #TrigAlarm_KA OR NOT #TrigAlarm_CCA1 OR NOT #TrigAlarm_CCA2;
END_REGION

REGION Network 39: Skip = Skip Alarm
   IF (#AlarmNo = 0) AND NOT #ALARM_AlarmPresent AND NOT #ALARM_FailureAckRequired THEN GOTO Skip; END_IF;
END_REGION

REGION Network 40: Clr = Clear Alarm
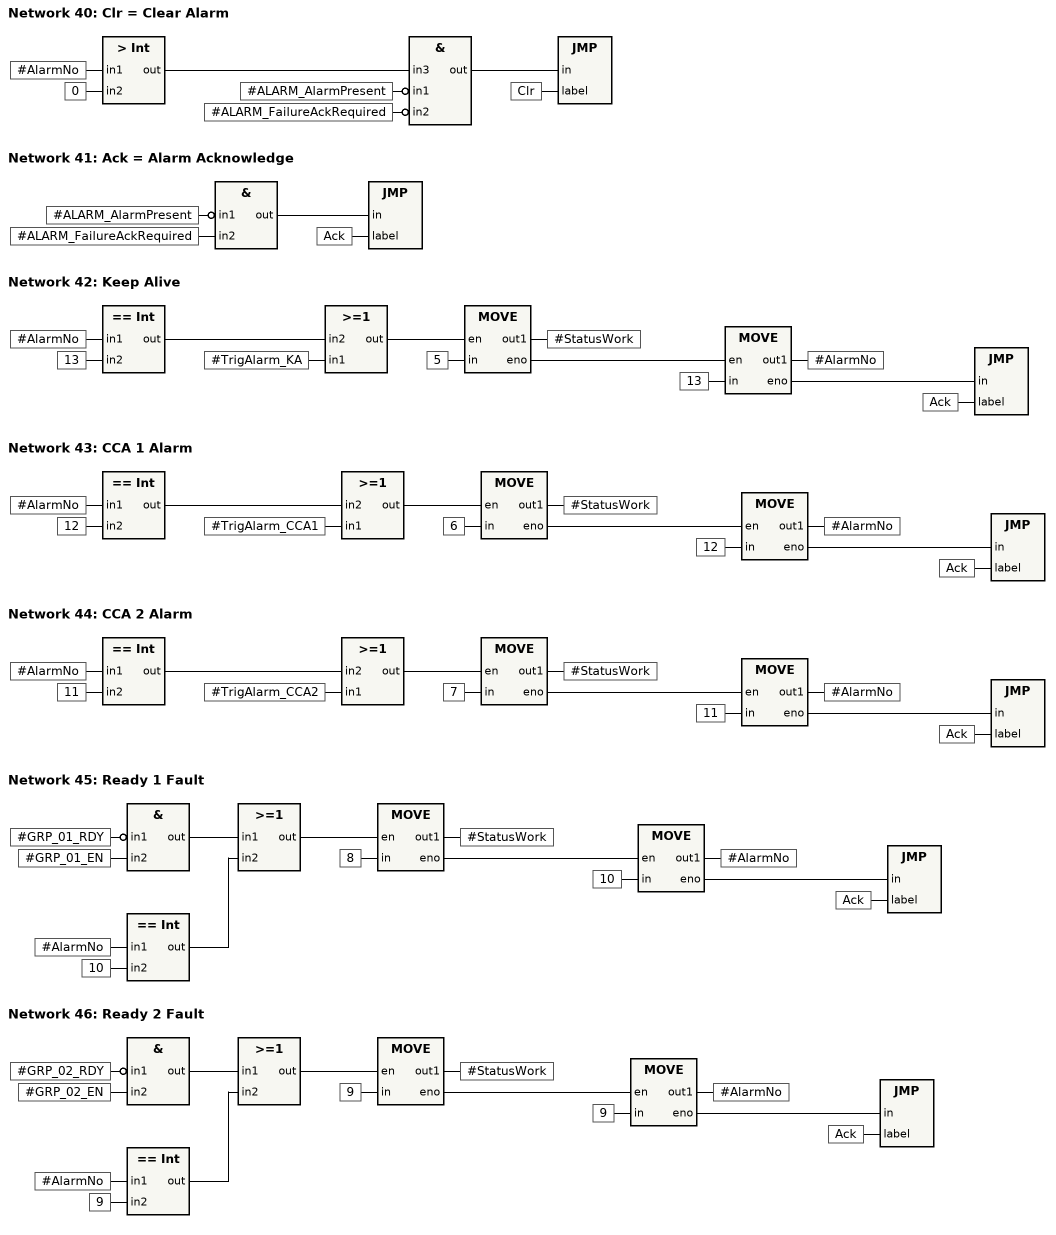
   IF (#AlarmNo > 0) AND NOT #ALARM_AlarmPresent AND NOT #ALARM_FailureAckRequired THEN GOTO Clr; END_IF;
END_REGION

REGION Network 41: Ack = Alarm Acknowledge
   IF NOT #ALARM_AlarmPresent AND #ALARM_FailureAckRequired THEN GOTO Ack; END_IF;
END_REGION

REGION Network 42: Keep Alive
   // ENO of a box is taken as its EN; it also drops when the box reports an error
   #_w1 := (#AlarmNo = 13) OR #TrigAlarm_KA;
   IF #_w1 THEN
       #StatusWork := 5;
       #AlarmNo := 13;
       GOTO Ack;
   END_IF;
END_REGION

REGION Network 43: CCA 1 Alarm
   // ENO of a box is taken as its EN; it also drops when the box reports an error
   #_w1 := (#AlarmNo = 12) OR #TrigAlarm_CCA1;
   IF #_w1 THEN
       #StatusWork := 6;
       #AlarmNo := 12;
       GOTO Ack;
   END_IF;
END_REGION

REGION Network 44: CCA 2 Alarm
   // ENO of a box is taken as its EN; it also drops when the box reports an error
   #_w1 := (#AlarmNo = 11) OR #TrigAlarm_CCA2;
   IF #_w1 THEN
       #StatusWork := 7;
       #AlarmNo := 11;
       GOTO Ack;
   END_IF;
END_REGION

REGION Network 45: Ready 1 Fault
   // ENO of a box is taken as its EN; it also drops when the box reports an error
   #_w1 := (NOT #GRP_01_RDY AND #GRP_01_EN) OR (#AlarmNo = 10);
   IF #_w1 THEN
       #StatusWork := 8;
       #AlarmNo := 10;
       GOTO Ack;
   END_IF;
END_REGION

REGION Network 46: Ready 2 Fault
   // ENO of a box is taken as its EN; it also drops when the box reports an error
   #_w1 := (NOT #GRP_02_RDY AND #GRP_02_EN) OR (#AlarmNo = 9);
   IF #_w1 THEN
       #StatusWork := 9;
       #AlarmNo := 9;
       GOTO Ack;
   END_IF;
END_REGION

REGION Network 47: Ready 3 Fault
